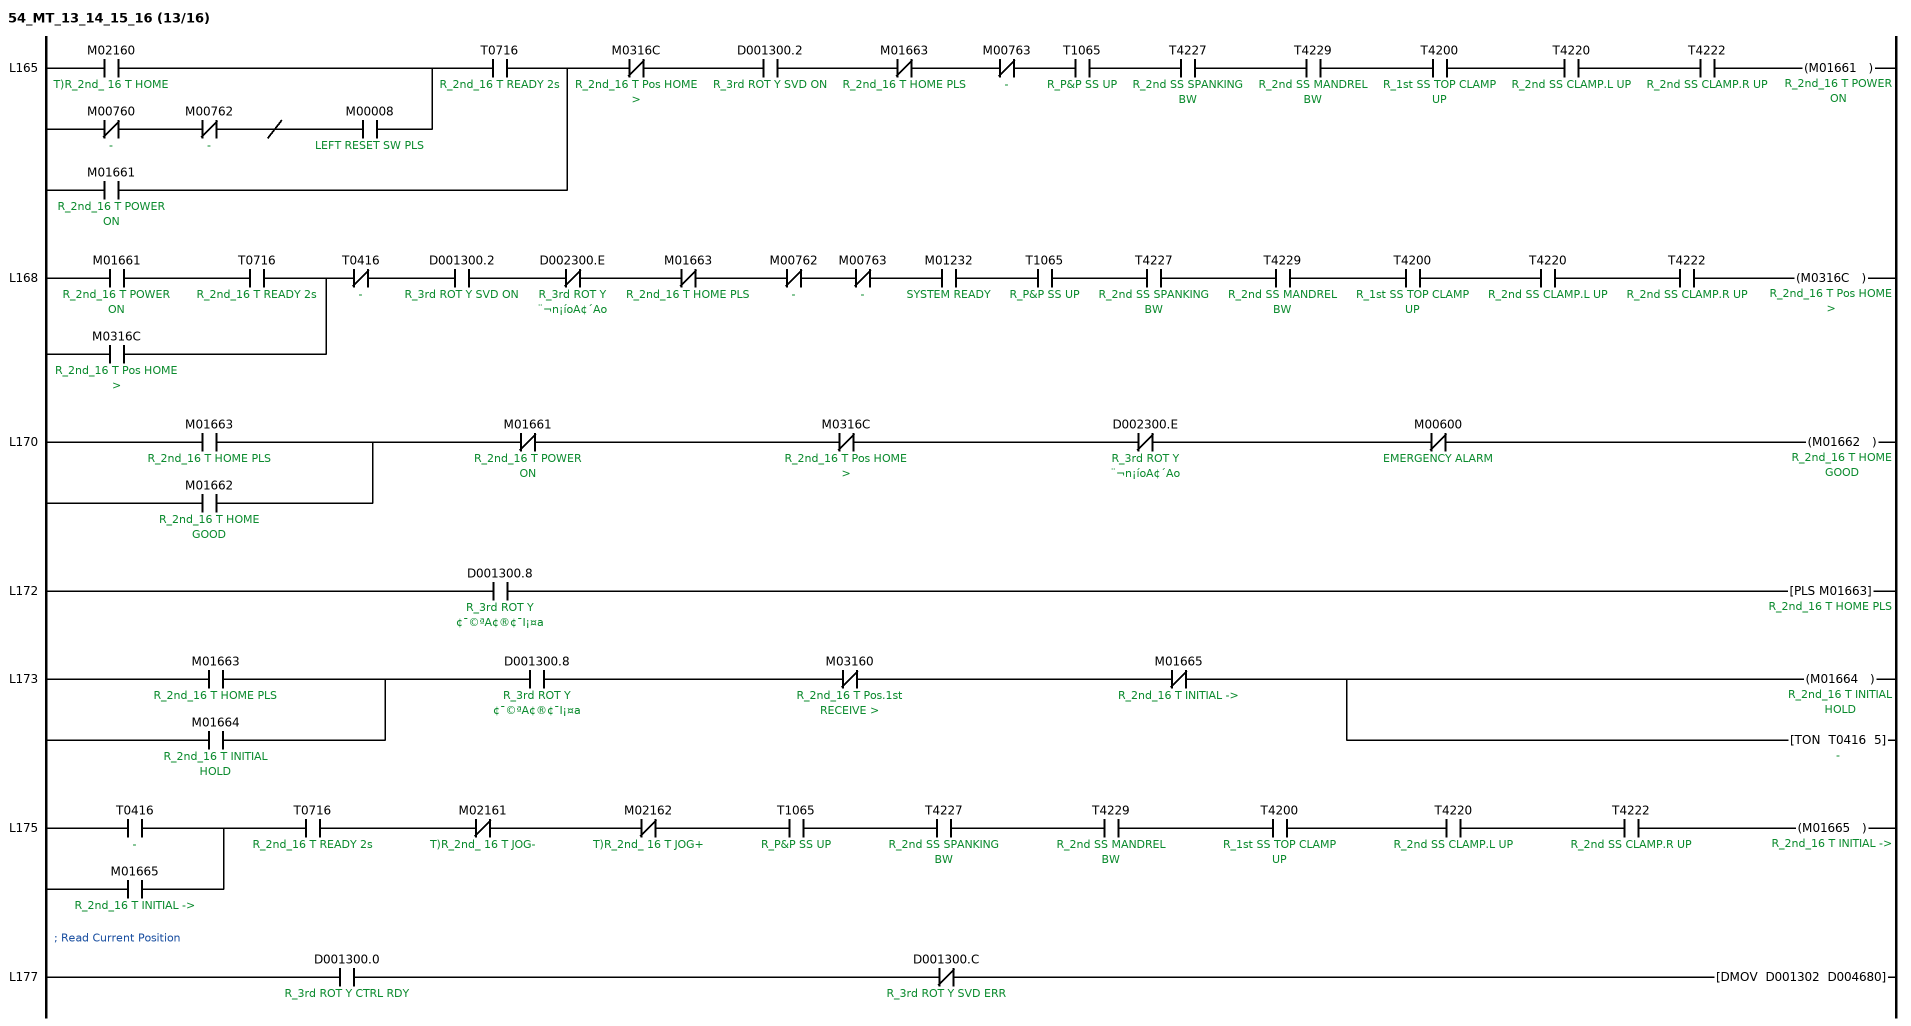
[picture p312: 54_MT_13_14_15_16 rungs L165-L177]
; L165
LOAD      M02160	// T)R_2nd_ 16 T HOME
LOAD NOT  M00760	// -
AND NOT   M00762	// -
NOT
AND       M00008	// LEFT RESET SW PLS
OR LOAD
AND       T0716	// R_2nd_16 T READY 2s
OR        M01661	// R_2nd_16 T POWER ON
AND NOT   M0316C	// R_2nd_16 T Pos HOME >
AND       D001300.2	// R_3rd ROT Y SVD ON
AND NOT   M01663	// R_2nd_16 T HOME PLS
AND NOT   M00763	// -
AND       T1065	// R_P&P SS UP
AND       T4227	// R_2nd SS SPANKING BW
AND       T4229	// R_2nd SS MANDREL BW
AND       T4200	// R_1st SS TOP CLAMP UP
AND       T4220	// R_2nd SS CLAMP.L UP
AND       T4222	// R_2nd SS CLAMP.R UP
OUT       M01661	// R_2nd_16 T POWER ON
; L168
LOAD      M01661	// R_2nd_16 T POWER ON
AND       T0716	// R_2nd_16 T READY 2s
OR        M0316C	// R_2nd_16 T Pos HOME >
AND NOT   T0416	// -
AND       D001300.2	// R_3rd ROT Y SVD ON
AND NOT   D002300.E	// R_3rd ROT Y ¨¬n¡íoA¢´Ao
AND NOT   M01663	// R_2nd_16 T HOME PLS
AND NOT   M00762	// -
AND NOT   M00763	// -
AND       M01232	// SYSTEM READY
AND       T1065	// R_P&P SS UP
AND       T4227	// R_2nd SS SPANKING BW
AND       T4229	// R_2nd SS MANDREL BW
AND       T4200	// R_1st SS TOP CLAMP UP
AND       T4220	// R_2nd SS CLAMP.L UP
AND       T4222	// R_2nd SS CLAMP.R UP
OUT       M0316C	// R_2nd_16 T Pos HOME >
; L170
LOAD      M01663	// R_2nd_16 T HOME PLS
OR        M01662	// R_2nd_16 T HOME GOOD
AND NOT   M01661	// R_2nd_16 T POWER ON
AND NOT   M0316C	// R_2nd_16 T Pos HOME >
AND NOT   D002300.E	// R_3rd ROT Y ¨¬n¡íoA¢´Ao
AND NOT   M00600	// EMERGENCY ALARM
OUT       M01662	// R_2nd_16 T HOME GOOD
; L172
LOAD      D001300.8	// R_3rd ROT Y ¢¯©ªA¢®¢¯I¡¤a
OUTP      M01663	// R_2nd_16 T HOME PLS
; L173
LOAD      M01663	// R_2nd_16 T HOME PLS
OR        M01664	// R_2nd_16 T INITIAL HOLD
AND       D001300.8	// R_3rd ROT Y ¢¯©ªA¢®¢¯I¡¤a
AND NOT   M03160	// R_2nd_16 T Pos.1st RECEIVE >
AND NOT   M01665	// R_2nd_16 T INITIAL ->
OUT       M01664	// R_2nd_16 T INITIAL HOLD
TON       T0416 5	// -
; L175
LOAD      T0416	// -
OR        M01665	// R_2nd_16 T INITIAL ->
AND       T0716	// R_2nd_16 T READY 2s
AND NOT   M02161	// T)R_2nd_ 16 T JOG-
AND NOT   M02162	// T)R_2nd_ 16 T JOG+
AND       T1065	// R_P&P SS UP
AND       T4227	// R_2nd SS SPANKING BW
AND       T4229	// R_2nd SS MANDREL BW
AND       T4200	// R_1st SS TOP CLAMP UP
AND       T4220	// R_2nd SS CLAMP.L UP
AND       T4222	// R_2nd SS CLAMP.R UP
OUT       M01665	// R_2nd_16 T INITIAL ->
; L177
LOAD      D001300.0	// R_3rd ROT Y CTRL RDY
AND NOT   D001300.C	// R_3rd ROT Y SVD ERR
DMOV      D001302 D004680
// output comment: Read Current Position

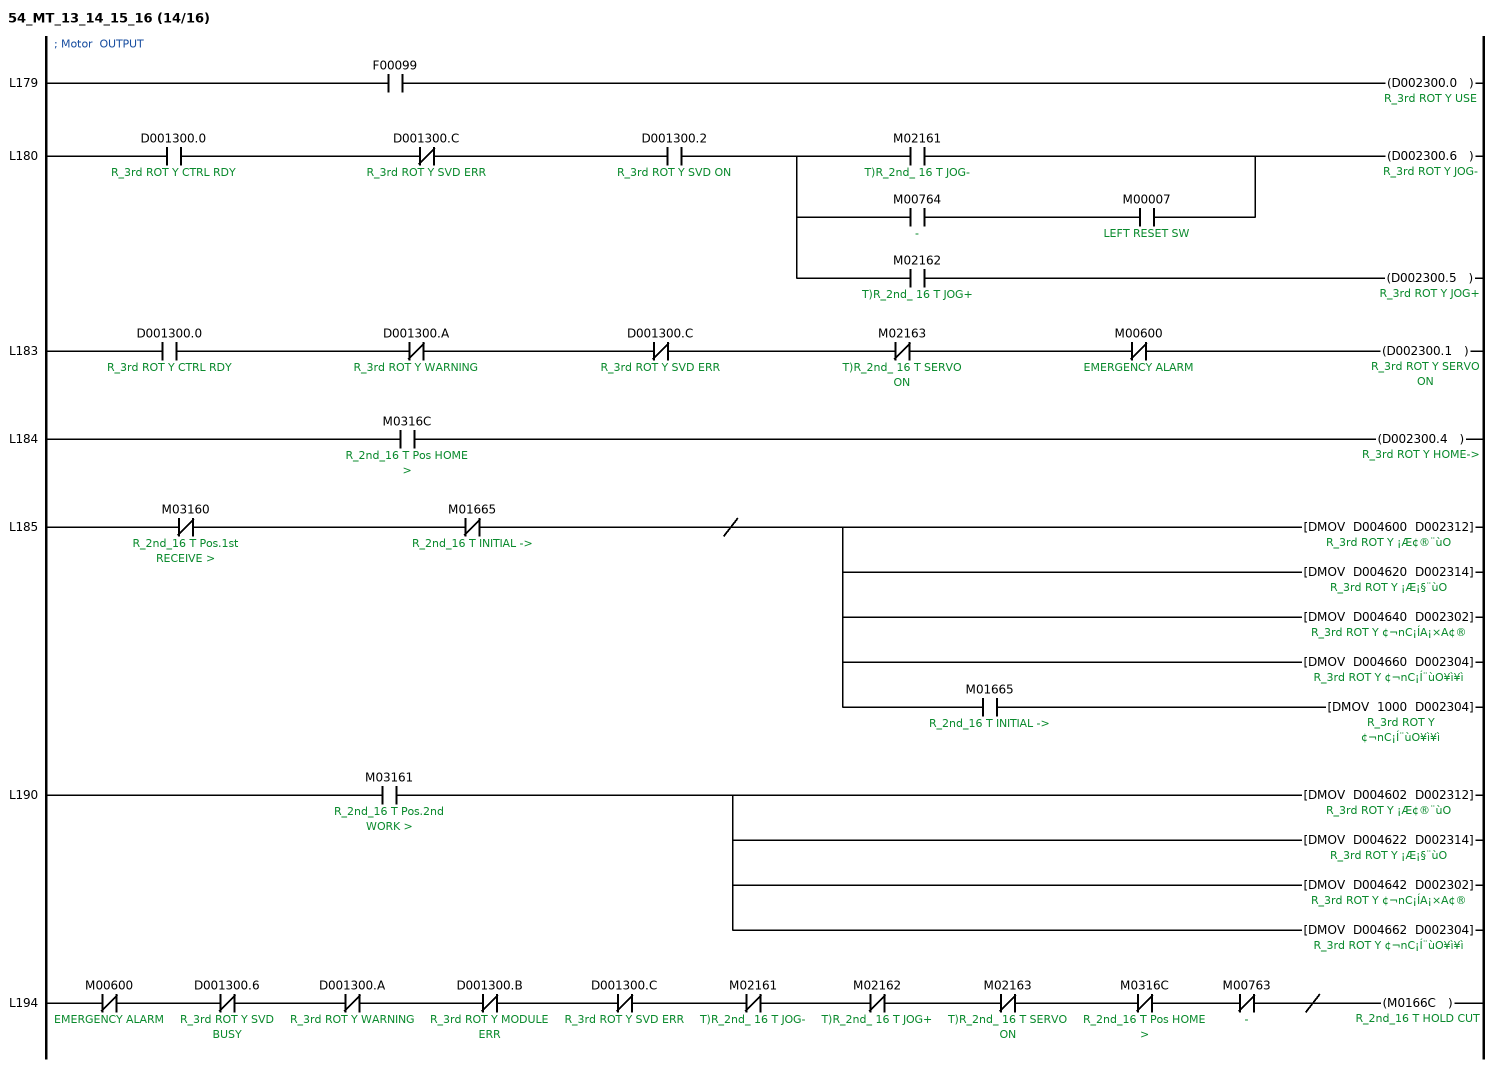
//  Motor  OUTPUT
; L179
LOAD      F00099
OUT       D002300.0	// R_3rd ROT Y USE
; L180
LOAD      D001300.0	// R_3rd ROT Y CTRL RDY
AND NOT   D001300.C	// R_3rd ROT Y SVD ERR
AND       D001300.2	// R_3rd ROT Y SVD ON
MPUSH
LOAD      M02161	// T)R_2nd_ 16 T JOG-
LOAD      M00764	// -
AND       M00007	// LEFT RESET SW
OR LOAD
AND LOAD
OUT       D002300.6	// R_3rd ROT Y JOG-
MPOP
AND       M02162	// T)R_2nd_ 16 T JOG+
OUT       D002300.5	// R_3rd ROT Y JOG+
; L183
LOAD      D001300.0	// R_3rd ROT Y CTRL RDY
AND NOT   D001300.A	// R_3rd ROT Y WARNING
AND NOT   D001300.C	// R_3rd ROT Y SVD ERR
AND NOT   M02163	// T)R_2nd_ 16 T SERVO ON
AND NOT   M00600	// EMERGENCY ALARM
OUT       D002300.1	// R_3rd ROT Y SERVO ON
; L184
LOAD      M0316C	// R_2nd_16 T Pos HOME >
OUT       D002300.4	// R_3rd ROT Y HOME->
; L185
LOAD NOT  M03160	// R_2nd_16 T Pos.1st RECEIVE >
AND NOT   M01665	// R_2nd_16 T INITIAL ->
NOT
DMOV      D004600 D002312	// R_3rd ROT Y ¡Æ¢®¨ùO
DMOV      D004620 D002314	// R_3rd ROT Y ¡Æ¡§¨ùO
DMOV      D004640 D002302	// R_3rd ROT Y ¢¬nC¡ÍA¡×A¢®
DMOV      D004660 D002304	// R_3rd ROT Y ¢¬nC¡Í¨ùO¥ì¥ì
AND       M01665	// R_2nd_16 T INITIAL ->
DMOV      1000 D002304	// R_3rd ROT Y ¢¬nC¡Í¨ùO¥ì¥ì
; L190
LOAD      M03161	// R_2nd_16 T Pos.2nd WORK >
DMOV      D004602 D002312	// R_3rd ROT Y ¡Æ¢®¨ùO
DMOV      D004622 D002314	// R_3rd ROT Y ¡Æ¡§¨ùO
DMOV      D004642 D002302	// R_3rd ROT Y ¢¬nC¡ÍA¡×A¢®
DMOV      D004662 D002304	// R_3rd ROT Y ¢¬nC¡Í¨ùO¥ì¥ì
; L194
LOAD NOT  M00600	// EMERGENCY ALARM
AND NOT   D001300.6	// R_3rd ROT Y SVD BUSY
AND NOT   D001300.A	// R_3rd ROT Y WARNING
AND NOT   D001300.B	// R_3rd ROT Y MODULE ERR
AND NOT   D001300.C	// R_3rd ROT Y SVD ERR
AND NOT   M02161	// T)R_2nd_ 16 T JOG-
AND NOT   M02162	// T)R_2nd_ 16 T JOG+
AND NOT   M02163	// T)R_2nd_ 16 T SERVO ON
AND NOT   M0316C	// R_2nd_16 T Pos HOME >
AND NOT   M00763	// -
NOT
OUT       M0166C	// R_2nd_16 T HOLD CUT

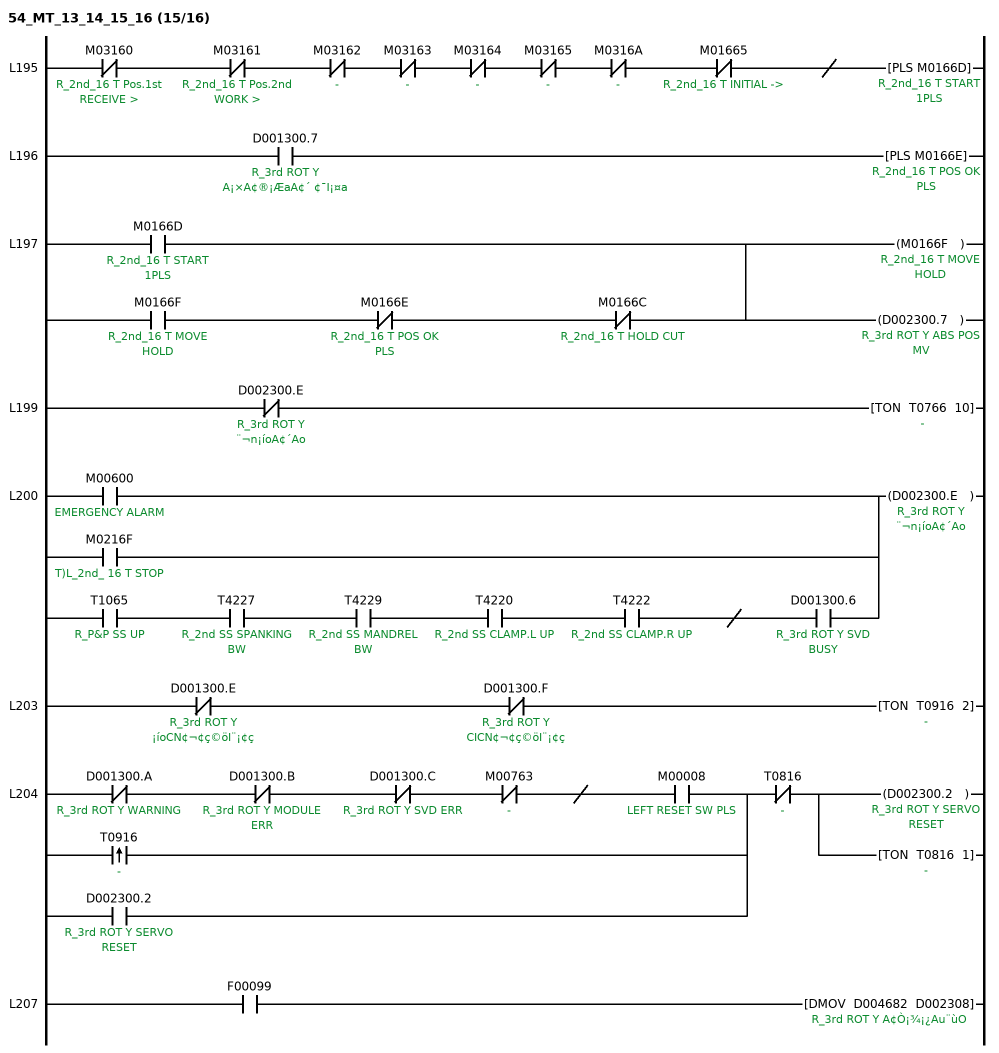
; L195
LOAD NOT  M03160	// R_2nd_16 T Pos.1st RECEIVE >
AND NOT   M03161	// R_2nd_16 T Pos.2nd WORK >
AND NOT   M03162	// -
AND NOT   M03163	// -
AND NOT   M03164	// -
AND NOT   M03165	// -
AND NOT   M0316A	// -
AND NOT   M01665	// R_2nd_16 T INITIAL ->
NOT
OUTP      M0166D	// R_2nd_16 T START 1PLS
; L196
LOAD      D001300.7	// R_3rd ROT Y A¡×A¢®¡ÆaA¢´ ¢¯I¡¤a
OUTP      M0166E	// R_2nd_16 T POS OK PLS
; L197
LOAD      M0166D	// R_2nd_16 T START 1PLS
LOAD      M0166F	// R_2nd_16 T MOVE HOLD
AND NOT   M0166E	// R_2nd_16 T POS OK PLS
AND NOT   M0166C	// R_2nd_16 T HOLD CUT
OR LOAD
OUT       M0166F	// R_2nd_16 T MOVE HOLD
OUT       D002300.7	// R_3rd ROT Y ABS POS MV
; L199
LOAD NOT  D002300.E	// R_3rd ROT Y ¨¬n¡íoA¢´Ao
TON       T0766 10	// -
; L200
LOAD      M00600	// EMERGENCY ALARM
OR        M0216F	// T)L_2nd_ 16 T STOP
LOAD      T1065	// R_P&P SS UP
AND       T4227	// R_2nd SS SPANKING BW
AND       T4229	// R_2nd SS MANDREL BW
AND       T4220	// R_2nd SS CLAMP.L UP
AND       T4222	// R_2nd SS CLAMP.R UP
NOT
AND       D001300.6	// R_3rd ROT Y SVD BUSY
OR LOAD
OUT       D002300.E	// R_3rd ROT Y ¨¬n¡íoA¢´Ao
; L203
LOAD NOT  D001300.E	// R_3rd ROT Y ¡íoCN¢¬¢ç©öI¨¡¢ç
AND NOT   D001300.F	// R_3rd ROT Y CICN¢¬¢ç©öI¨¡¢ç
TON       T0916 2	// -
; L204
LOAD NOT  D001300.A	// R_3rd ROT Y WARNING
AND NOT   D001300.B	// R_3rd ROT Y MODULE ERR
AND NOT   D001300.C	// R_3rd ROT Y SVD ERR
AND NOT   M00763	// -
NOT
AND       M00008	// LEFT RESET SW PLS
ORP       T0916	// -
OR        D002300.2	// R_3rd ROT Y SERVO RESET
AND NOT   T0816	// -
OUT       D002300.2	// R_3rd ROT Y SERVO RESET
TON       T0816 1	// -
; L207
LOAD      F00099
DMOV      D004682 D002308	// R_3rd ROT Y A¢Ò¡¾¡¿Au¨ùO

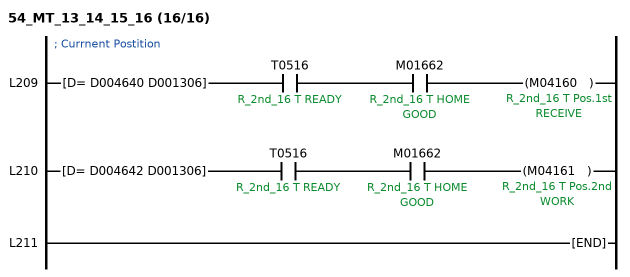
// Currnent Postition
; L209
LOADD=    D004640 D001306
AND       T0516	// R_2nd_16 T READY
AND       M01662	// R_2nd_16 T HOME GOOD
OUT       M04160	// R_2nd_16 T Pos.1st RECEIVE
; L210
LOADD=    D004642 D001306
AND       T0516	// R_2nd_16 T READY
AND       M01662	// R_2nd_16 T HOME GOOD
OUT       M04161	// R_2nd_16 T Pos.2nd WORK
; L211
END

PROGRAM 55_MT_17_18_19_20 (task: ¨ö¨¬A¥ì CA¡¤I¡¾¡¿¡¤¡Í)

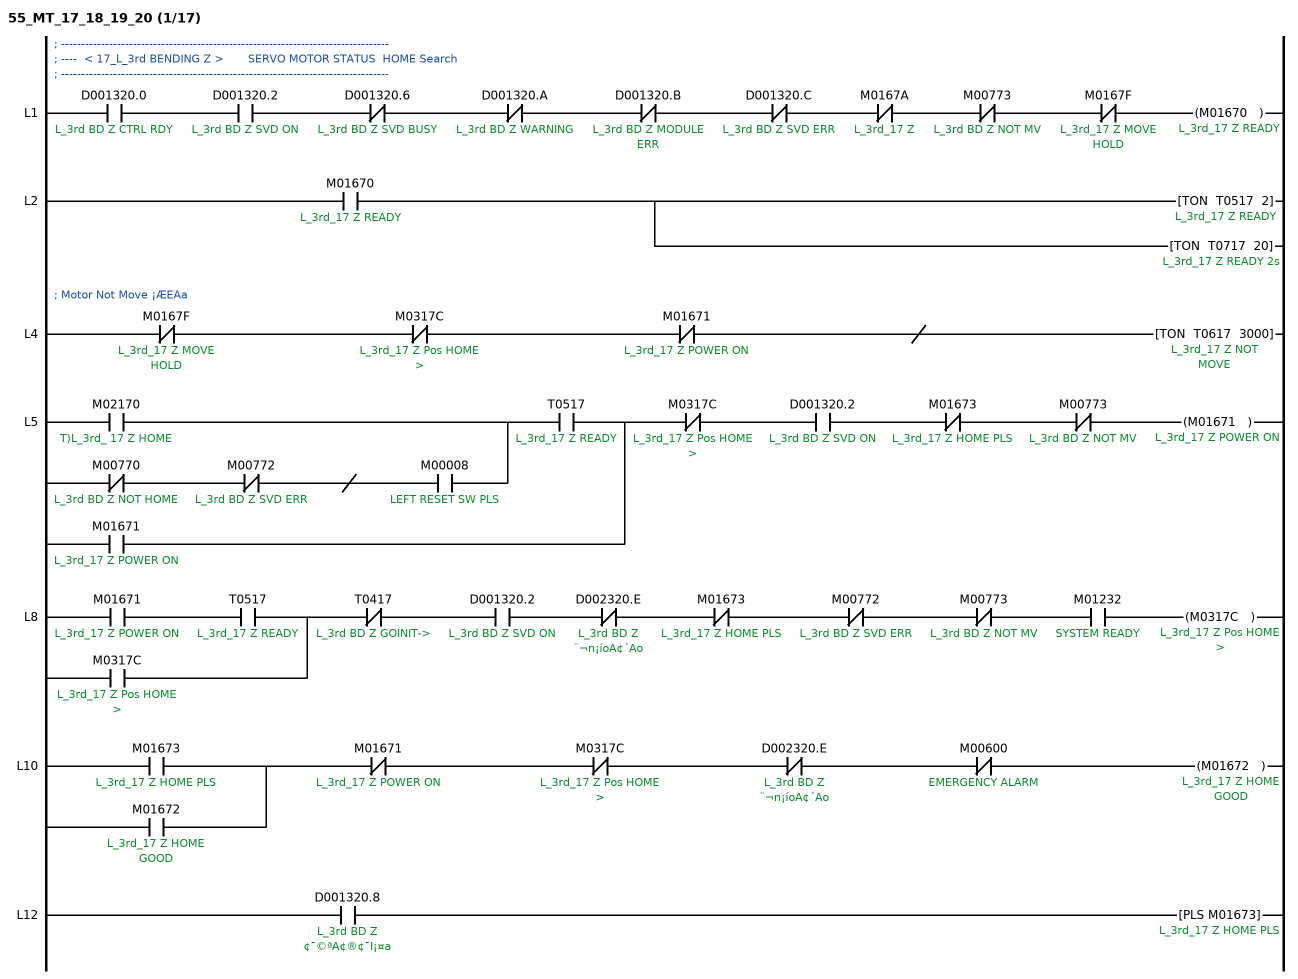
// ----------------------------------------------------------------------------------
// 
// ----  < 17_L_3rd BENDING Z >       SERVO MOTOR STATUS  HOME Search
// 
// ----------------------------------------------------------------------------------
; L1
LOAD      D001320.0	// L_3rd BD Z CTRL RDY
AND       D001320.2	// L_3rd BD Z SVD ON
AND NOT   D001320.6	// L_3rd BD Z SVD BUSY
AND NOT   D001320.A	// L_3rd BD Z WARNING
AND NOT   D001320.B	// L_3rd BD Z MODULE ERR
AND NOT   D001320.C	// L_3rd BD Z SVD ERR
AND NOT   M0167A	// L_3rd_17 Z
AND NOT   M00773	// L_3rd BD Z NOT MV
AND NOT   M0167F	// L_3rd_17 Z MOVE HOLD
OUT       M01670	// L_3rd_17 Z READY
; L2
LOAD      M01670	// L_3rd_17 Z READY
TON       T0517 2	// L_3rd_17 Z READY
TON       T0717 20	// L_3rd_17 Z READY 2s
; L4
LOAD NOT  M0167F	// L_3rd_17 Z MOVE HOLD
AND NOT   M0317C	// L_3rd_17 Z Pos HOME >
AND NOT   M01671	// L_3rd_17 Z POWER ON
NOT
TON       T0617 3000	// L_3rd_17 Z NOT MOVE
// output comment: Motor Not Move ¡ÆEAa
; L5
LOAD      M02170	// T)L_3rd_ 17 Z HOME
LOAD NOT  M00770	// L_3rd BD Z NOT HOME
AND NOT   M00772	// L_3rd BD Z SVD ERR
NOT
AND       M00008	// LEFT RESET SW PLS
OR LOAD
AND       T0517	// L_3rd_17 Z READY
OR        M01671	// L_3rd_17 Z POWER ON
AND NOT   M0317C	// L_3rd_17 Z Pos HOME >
AND       D001320.2	// L_3rd BD Z SVD ON
AND NOT   M01673	// L_3rd_17 Z HOME PLS
AND NOT   M00773	// L_3rd BD Z NOT MV
OUT       M01671	// L_3rd_17 Z POWER ON
; L8
LOAD      M01671	// L_3rd_17 Z POWER ON
AND       T0517	// L_3rd_17 Z READY
OR        M0317C	// L_3rd_17 Z Pos HOME >
AND NOT   T0417	// L_3rd BD Z GOINIT->
AND       D001320.2	// L_3rd BD Z SVD ON
AND NOT   D002320.E	// L_3rd BD Z ¨¬n¡íoA¢´Ao
AND NOT   M01673	// L_3rd_17 Z HOME PLS
AND NOT   M00772	// L_3rd BD Z SVD ERR
AND NOT   M00773	// L_3rd BD Z NOT MV
AND       M01232	// SYSTEM READY
OUT       M0317C	// L_3rd_17 Z Pos HOME >
; L10
LOAD      M01673	// L_3rd_17 Z HOME PLS
OR        M01672	// L_3rd_17 Z HOME GOOD
AND NOT   M01671	// L_3rd_17 Z POWER ON
AND NOT   M0317C	// L_3rd_17 Z Pos HOME >
AND NOT   D002320.E	// L_3rd BD Z ¨¬n¡íoA¢´Ao
AND NOT   M00600	// EMERGENCY ALARM
OUT       M01672	// L_3rd_17 Z HOME GOOD
; L12
LOAD      D001320.8	// L_3rd BD Z ¢¯©ªA¢®¢¯I¡¤a
OUTP      M01673	// L_3rd_17 Z HOME PLS

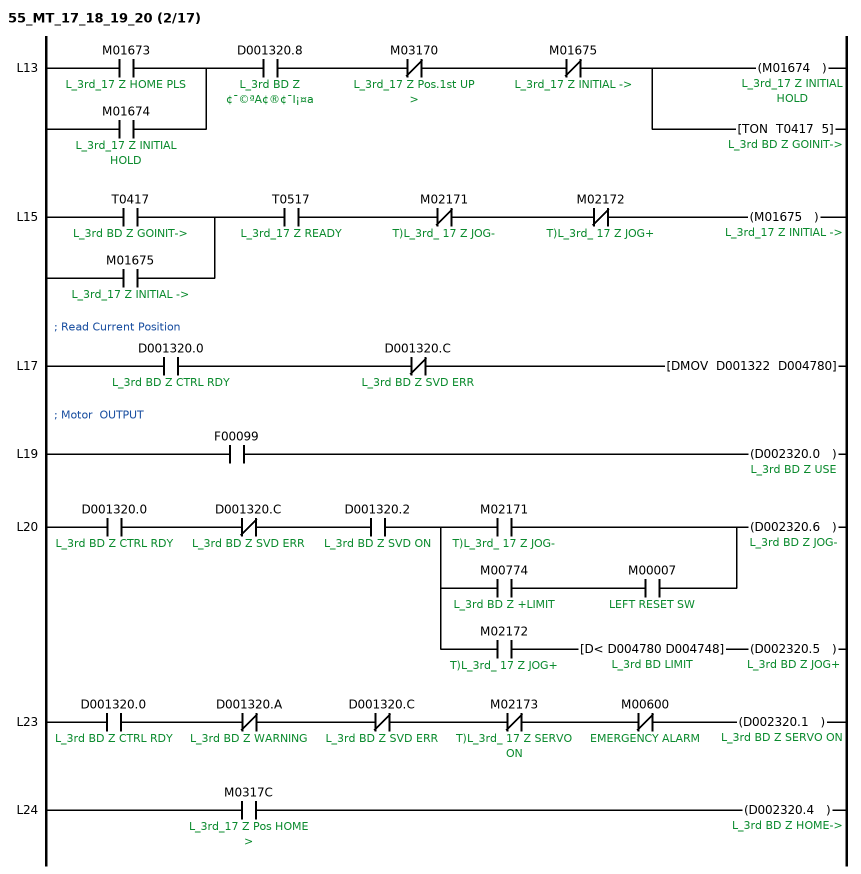
; L13
LOAD      M01673	// L_3rd_17 Z HOME PLS
OR        M01674	// L_3rd_17 Z INITIAL HOLD
AND       D001320.8	// L_3rd BD Z ¢¯©ªA¢®¢¯I¡¤a
AND NOT   M03170	// L_3rd_17 Z Pos.1st UP >
AND NOT   M01675	// L_3rd_17 Z INITIAL ->
OUT       M01674	// L_3rd_17 Z INITIAL HOLD
TON       T0417 5	// L_3rd BD Z GOINIT->
; L15
LOAD      T0417	// L_3rd BD Z GOINIT->
OR        M01675	// L_3rd_17 Z INITIAL ->
AND       T0517	// L_3rd_17 Z READY
AND NOT   M02171	// T)L_3rd_ 17 Z JOG-
AND NOT   M02172	// T)L_3rd_ 17 Z JOG+
OUT       M01675	// L_3rd_17 Z INITIAL ->
; L17
LOAD      D001320.0	// L_3rd BD Z CTRL RDY
AND NOT   D001320.C	// L_3rd BD Z SVD ERR
DMOV      D001322 D004780
// output comment: Read Current Position
//  Motor  OUTPUT
; L19
LOAD      F00099
OUT       D002320.0	// L_3rd BD Z USE
; L20
LOAD      D001320.0	// L_3rd BD Z CTRL RDY
AND NOT   D001320.C	// L_3rd BD Z SVD ERR
AND       D001320.2	// L_3rd BD Z SVD ON
MPUSH
LOAD      M02171	// T)L_3rd_ 17 Z JOG-
LOAD      M00774	// L_3rd BD Z +LIMIT
AND       M00007	// LEFT RESET SW
OR LOAD
AND LOAD
OUT       D002320.6	// L_3rd BD Z JOG-
MPOP
AND       M02172	// T)L_3rd_ 17 Z JOG+
ANDD<     D004780 D004748	// L_3rd BD LIMIT
OUT       D002320.5	// L_3rd BD Z JOG+
; L23
LOAD      D001320.0	// L_3rd BD Z CTRL RDY
AND NOT   D001320.A	// L_3rd BD Z WARNING
AND NOT   D001320.C	// L_3rd BD Z SVD ERR
AND NOT   M02173	// T)L_3rd_ 17 Z SERVO ON
AND NOT   M00600	// EMERGENCY ALARM
OUT       D002320.1	// L_3rd BD Z SERVO ON
; L24
LOAD      M0317C	// L_3rd_17 Z Pos HOME >
OUT       D002320.4	// L_3rd BD Z HOME->

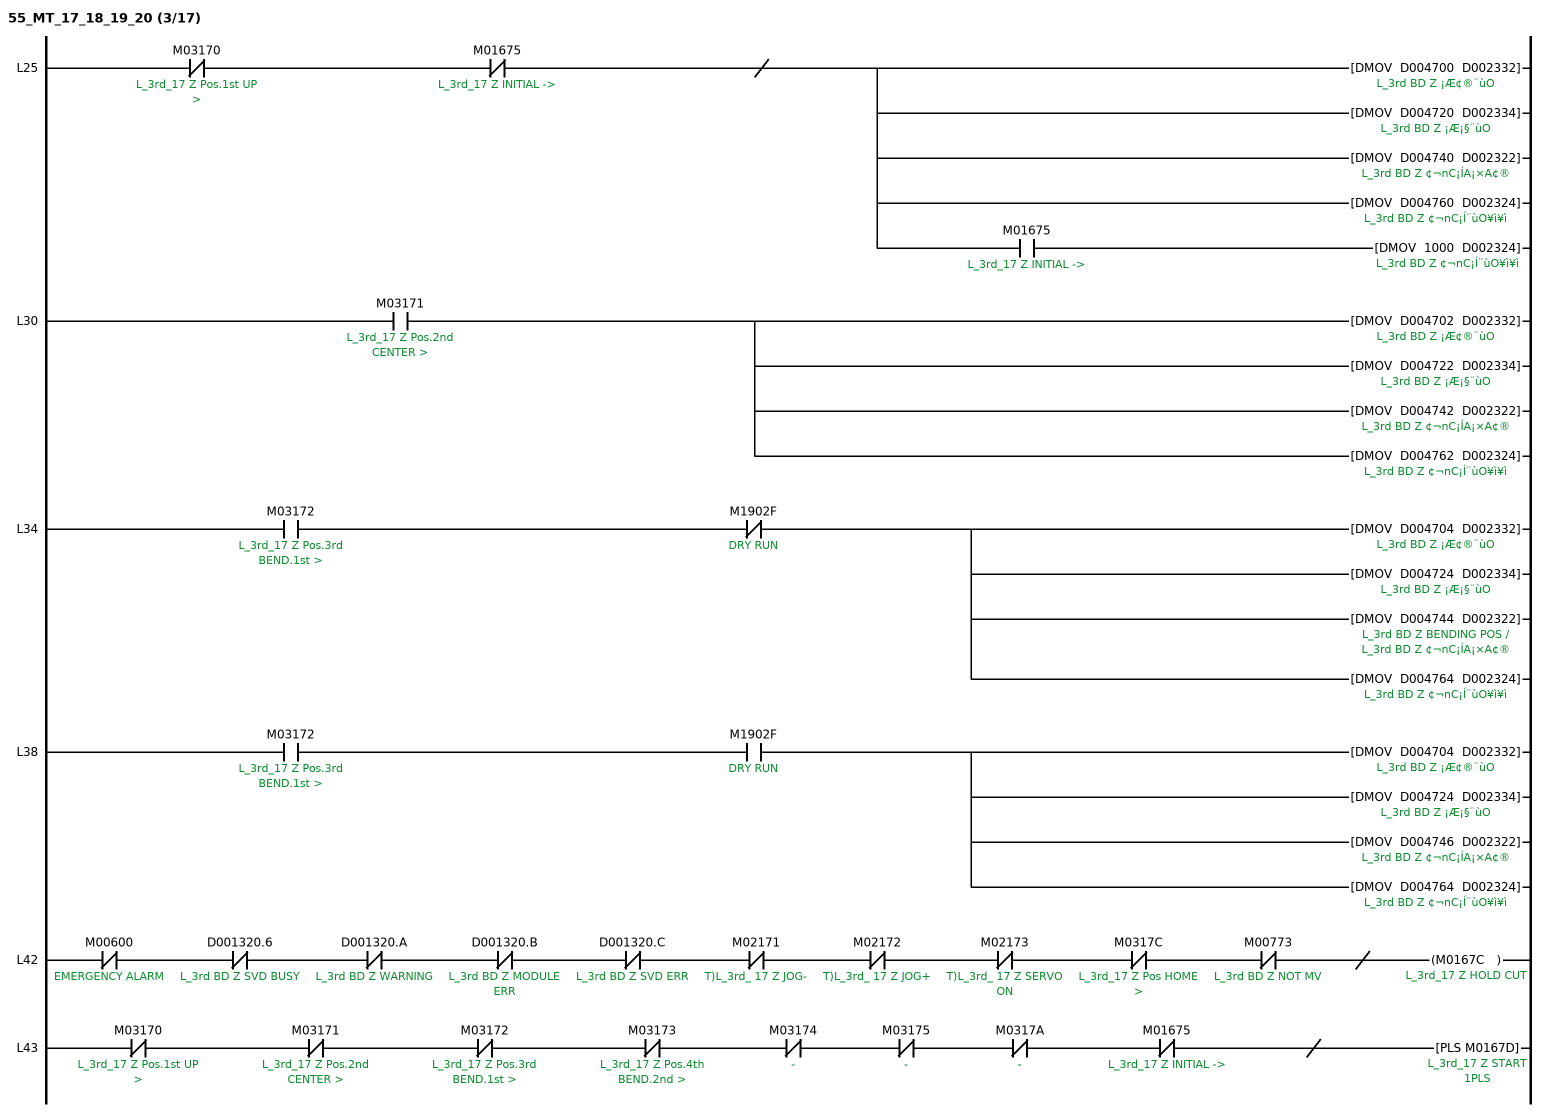
; L25
LOAD NOT  M03170	// L_3rd_17 Z Pos.1st UP >
AND NOT   M01675	// L_3rd_17 Z INITIAL ->
NOT
DMOV      D004700 D002332	// L_3rd BD Z ¡Æ¢®¨ùO
DMOV      D004720 D002334	// L_3rd BD Z ¡Æ¡§¨ùO
DMOV      D004740 D002322	// L_3rd BD Z ¢¬nC¡ÍA¡×A¢®
DMOV      D004760 D002324	// L_3rd BD Z ¢¬nC¡Í¨ùO¥ì¥ì
AND       M01675	// L_3rd_17 Z INITIAL ->
DMOV      1000 D002324	// L_3rd BD Z ¢¬nC¡Í¨ùO¥ì¥ì
; L30
LOAD      M03171	// L_3rd_17 Z Pos.2nd CENTER >
DMOV      D004702 D002332	// L_3rd BD Z ¡Æ¢®¨ùO
DMOV      D004722 D002334	// L_3rd BD Z ¡Æ¡§¨ùO
DMOV      D004742 D002322	// L_3rd BD Z ¢¬nC¡ÍA¡×A¢®
DMOV      D004762 D002324	// L_3rd BD Z ¢¬nC¡Í¨ùO¥ì¥ì
; L34
LOAD      M03172	// L_3rd_17 Z Pos.3rd BEND.1st >
AND NOT   M1902F	// DRY RUN
DMOV      D004704 D002332	// L_3rd BD Z ¡Æ¢®¨ùO
DMOV      D004724 D002334	// L_3rd BD Z ¡Æ¡§¨ùO
DMOV      D004744 D002322	// L_3rd BD Z BENDING POS / L_3rd BD Z ¢¬nC¡ÍA¡×A¢®
DMOV      D004764 D002324	// L_3rd BD Z ¢¬nC¡Í¨ùO¥ì¥ì
; L38
LOAD      M03172	// L_3rd_17 Z Pos.3rd BEND.1st >
AND       M1902F	// DRY RUN
DMOV      D004704 D002332	// L_3rd BD Z ¡Æ¢®¨ùO
DMOV      D004724 D002334	// L_3rd BD Z ¡Æ¡§¨ùO
DMOV      D004746 D002322	// L_3rd BD Z ¢¬nC¡ÍA¡×A¢®
DMOV      D004764 D002324	// L_3rd BD Z ¢¬nC¡Í¨ùO¥ì¥ì
; L42
LOAD NOT  M00600	// EMERGENCY ALARM
AND NOT   D001320.6	// L_3rd BD Z SVD BUSY
AND NOT   D001320.A	// L_3rd BD Z WARNING
AND NOT   D001320.B	// L_3rd BD Z MODULE ERR
AND NOT   D001320.C	// L_3rd BD Z SVD ERR
AND NOT   M02171	// T)L_3rd_ 17 Z JOG-
AND NOT   M02172	// T)L_3rd_ 17 Z JOG+
AND NOT   M02173	// T)L_3rd_ 17 Z SERVO ON
AND NOT   M0317C	// L_3rd_17 Z Pos HOME >
AND NOT   M00773	// L_3rd BD Z NOT MV
NOT
OUT       M0167C	// L_3rd_17 Z HOLD CUT
; L43
LOAD NOT  M03170	// L_3rd_17 Z Pos.1st UP >
AND NOT   M03171	// L_3rd_17 Z Pos.2nd CENTER >
AND NOT   M03172	// L_3rd_17 Z Pos.3rd BEND.1st >
AND NOT   M03173	// L_3rd_17 Z Pos.4th BEND.2nd >
AND NOT   M03174	// -
AND NOT   M03175	// -
AND NOT   M0317A	// -
AND NOT   M01675	// L_3rd_17 Z INITIAL ->
NOT
OUTP      M0167D	// L_3rd_17 Z START 1PLS

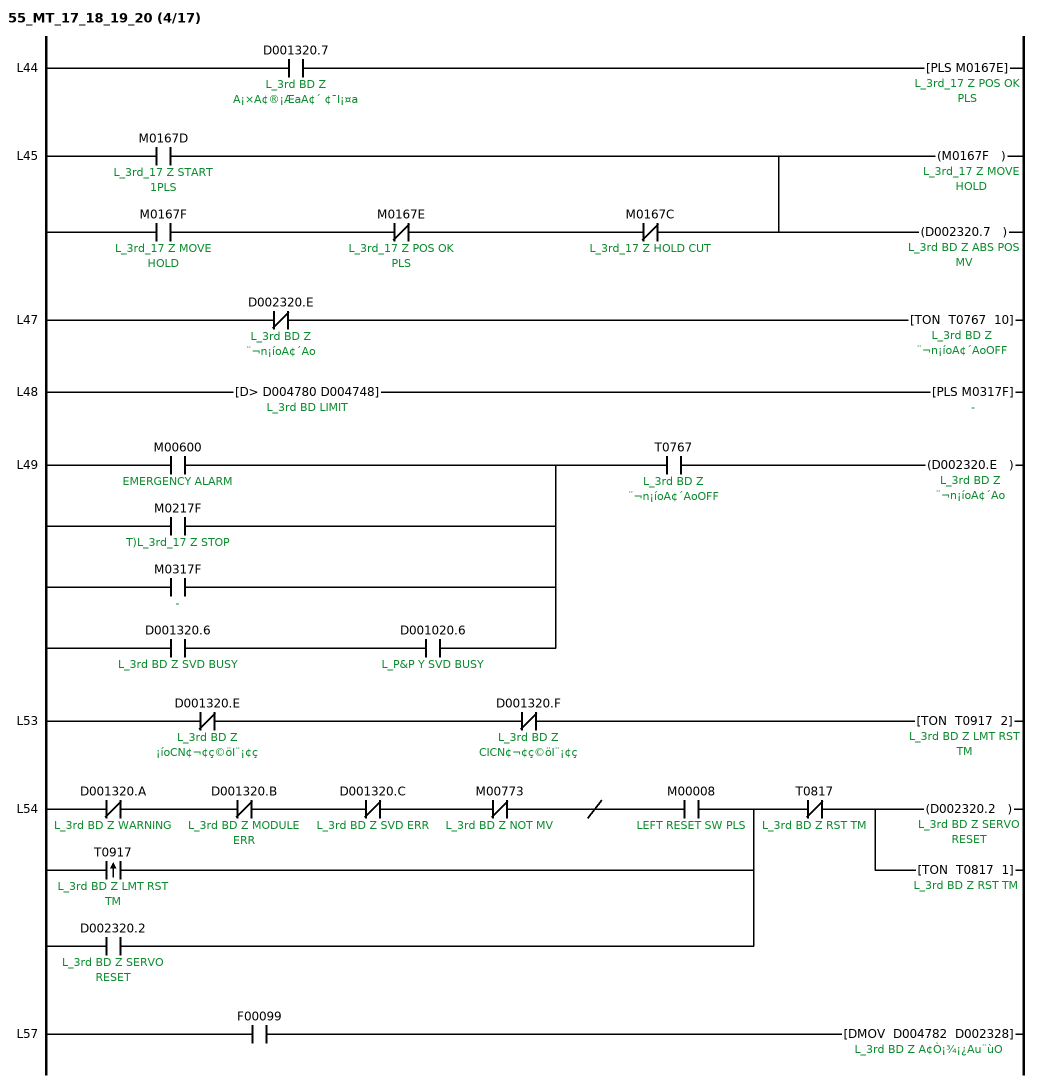
; L44
LOAD      D001320.7	// L_3rd BD Z A¡×A¢®¡ÆaA¢´ ¢¯I¡¤a
OUTP      M0167E	// L_3rd_17 Z POS OK PLS
; L45
LOAD      M0167D	// L_3rd_17 Z START 1PLS
LOAD      M0167F	// L_3rd_17 Z MOVE HOLD
AND NOT   M0167E	// L_3rd_17 Z POS OK PLS
AND NOT   M0167C	// L_3rd_17 Z HOLD CUT
OR LOAD
OUT       M0167F	// L_3rd_17 Z MOVE HOLD
OUT       D002320.7	// L_3rd BD Z ABS POS MV
; L47
LOAD NOT  D002320.E	// L_3rd BD Z ¨¬n¡íoA¢´Ao
TON       T0767 10	// L_3rd BD Z ¨¬n¡íoA¢´AoOFF
; L48
LOADD>    D004780 D004748	// L_3rd BD LIMIT
OUTP      M0317F	// -
; L49
LOAD      M00600	// EMERGENCY ALARM
OR        M0217F	// T)L_3rd_17 Z STOP
OR        M0317F	// -
LOAD      D001320.6	// L_3rd BD Z SVD BUSY
AND       D001020.6	// L_P&P Y SVD BUSY
OR LOAD
AND       T0767	// L_3rd BD Z ¨¬n¡íoA¢´AoOFF
OUT       D002320.E	// L_3rd BD Z ¨¬n¡íoA¢´Ao
; L53
LOAD NOT  D001320.E	// L_3rd BD Z ¡íoCN¢¬¢ç©öI¨¡¢ç
AND NOT   D001320.F	// L_3rd BD Z CICN¢¬¢ç©öI¨¡¢ç
TON       T0917 2	// L_3rd BD Z LMT RST TM
; L54
LOAD NOT  D001320.A	// L_3rd BD Z WARNING
AND NOT   D001320.B	// L_3rd BD Z MODULE ERR
AND NOT   D001320.C	// L_3rd BD Z SVD ERR
AND NOT   M00773	// L_3rd BD Z NOT MV
NOT
AND       M00008	// LEFT RESET SW PLS
ORP       T0917	// L_3rd BD Z LMT RST TM
OR        D002320.2	// L_3rd BD Z SERVO RESET
AND NOT   T0817	// L_3rd BD Z RST TM
OUT       D002320.2	// L_3rd BD Z SERVO RESET
TON       T0817 1	// L_3rd BD Z RST TM
; L57
LOAD      F00099
DMOV      D004782 D002328	// L_3rd BD Z A¢Ò¡¾¡¿Au¨ùO

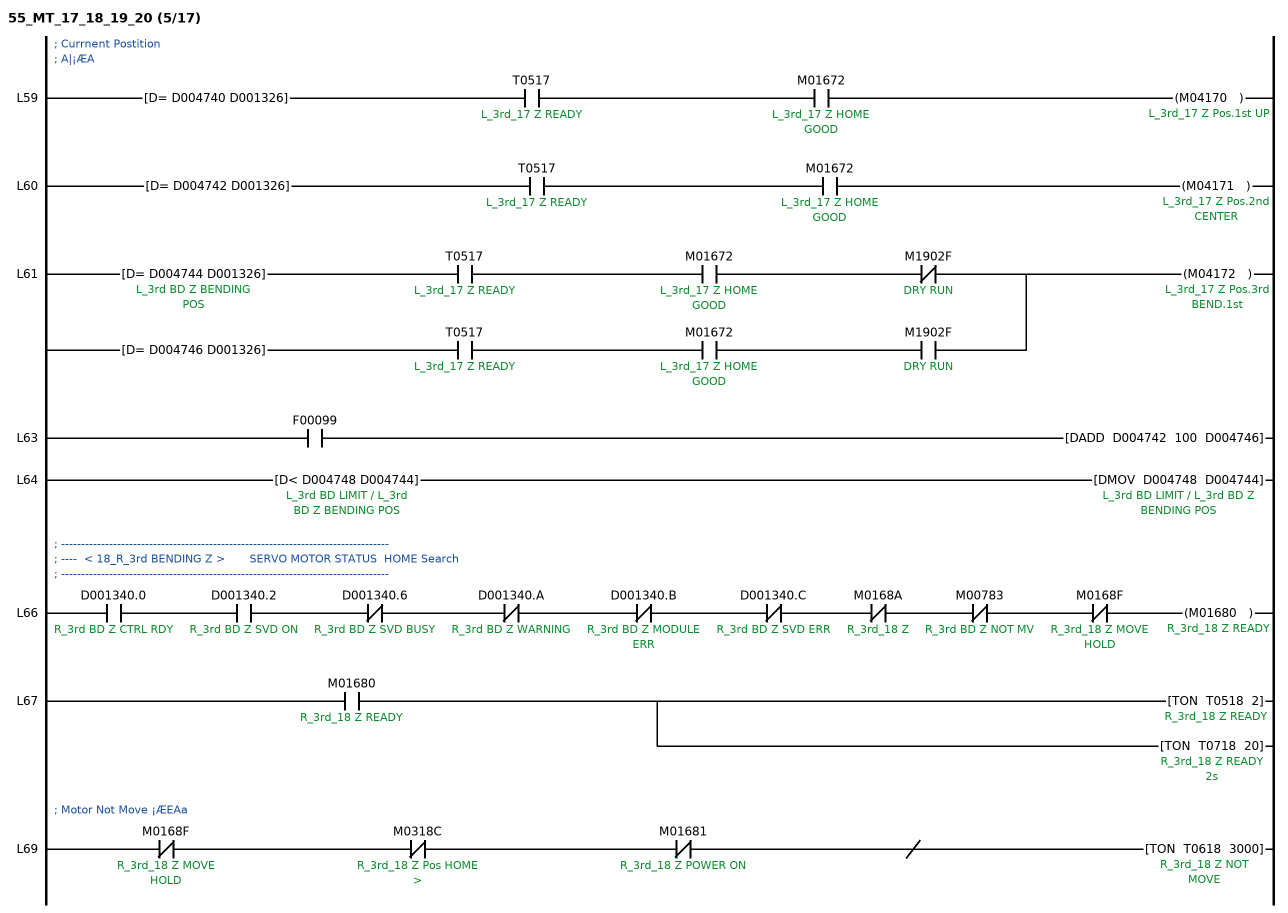
// Currnent Postition
; L59
LOADD=    D004740 D001326
AND       T0517	// L_3rd_17 Z READY
AND       M01672	// L_3rd_17 Z HOME GOOD
OUT       M04170	// L_3rd_17 Z Pos.1st UP
// output comment: A|¡ÆA
; L60
LOADD=    D004742 D001326
AND       T0517	// L_3rd_17 Z READY
AND       M01672	// L_3rd_17 Z HOME GOOD
OUT       M04171	// L_3rd_17 Z Pos.2nd CENTER
; L61
LOADD=    D004744 D001326	// L_3rd BD Z BENDING POS
AND       T0517	// L_3rd_17 Z READY
AND       M01672	// L_3rd_17 Z HOME GOOD
AND NOT   M1902F	// DRY RUN
LOADD=    D004746 D001326
AND       T0517	// L_3rd_17 Z READY
AND       M01672	// L_3rd_17 Z HOME GOOD
AND       M1902F	// DRY RUN
OR LOAD
OUT       M04172	// L_3rd_17 Z Pos.3rd BEND.1st
; L63
LOAD      F00099
DADD      D004742 100 D004746
; L64
LOADD<    D004748 D004744	// L_3rd BD LIMIT / L_3rd BD Z BENDING POS
DMOV      D004748 D004744	// L_3rd BD LIMIT / L_3rd BD Z BENDING POS
// ----------------------------------------------------------------------------------
// 
// ----  < 18_R_3rd BENDING Z >       SERVO MOTOR STATUS  HOME Search
// 
// ----------------------------------------------------------------------------------
; L66
LOAD      D001340.0	// R_3rd BD Z CTRL RDY
AND       D001340.2	// R_3rd BD Z SVD ON
AND NOT   D001340.6	// R_3rd BD Z SVD BUSY
AND NOT   D001340.A	// R_3rd BD Z WARNING
AND NOT   D001340.B	// R_3rd BD Z MODULE ERR
AND NOT   D001340.C	// R_3rd BD Z SVD ERR
AND NOT   M0168A	// R_3rd_18 Z
AND NOT   M00783	// R_3rd BD Z NOT MV
AND NOT   M0168F	// R_3rd_18 Z MOVE HOLD
OUT       M01680	// R_3rd_18 Z READY
; L67
LOAD      M01680	// R_3rd_18 Z READY
TON       T0518 2	// R_3rd_18 Z READY
TON       T0718 20	// R_3rd_18 Z READY 2s
; L69
LOAD NOT  M0168F	// R_3rd_18 Z MOVE HOLD
AND NOT   M0318C	// R_3rd_18 Z Pos HOME >
AND NOT   M01681	// R_3rd_18 Z POWER ON
NOT
TON       T0618 3000	// R_3rd_18 Z NOT MOVE
// output comment: Motor Not Move ¡ÆEAa

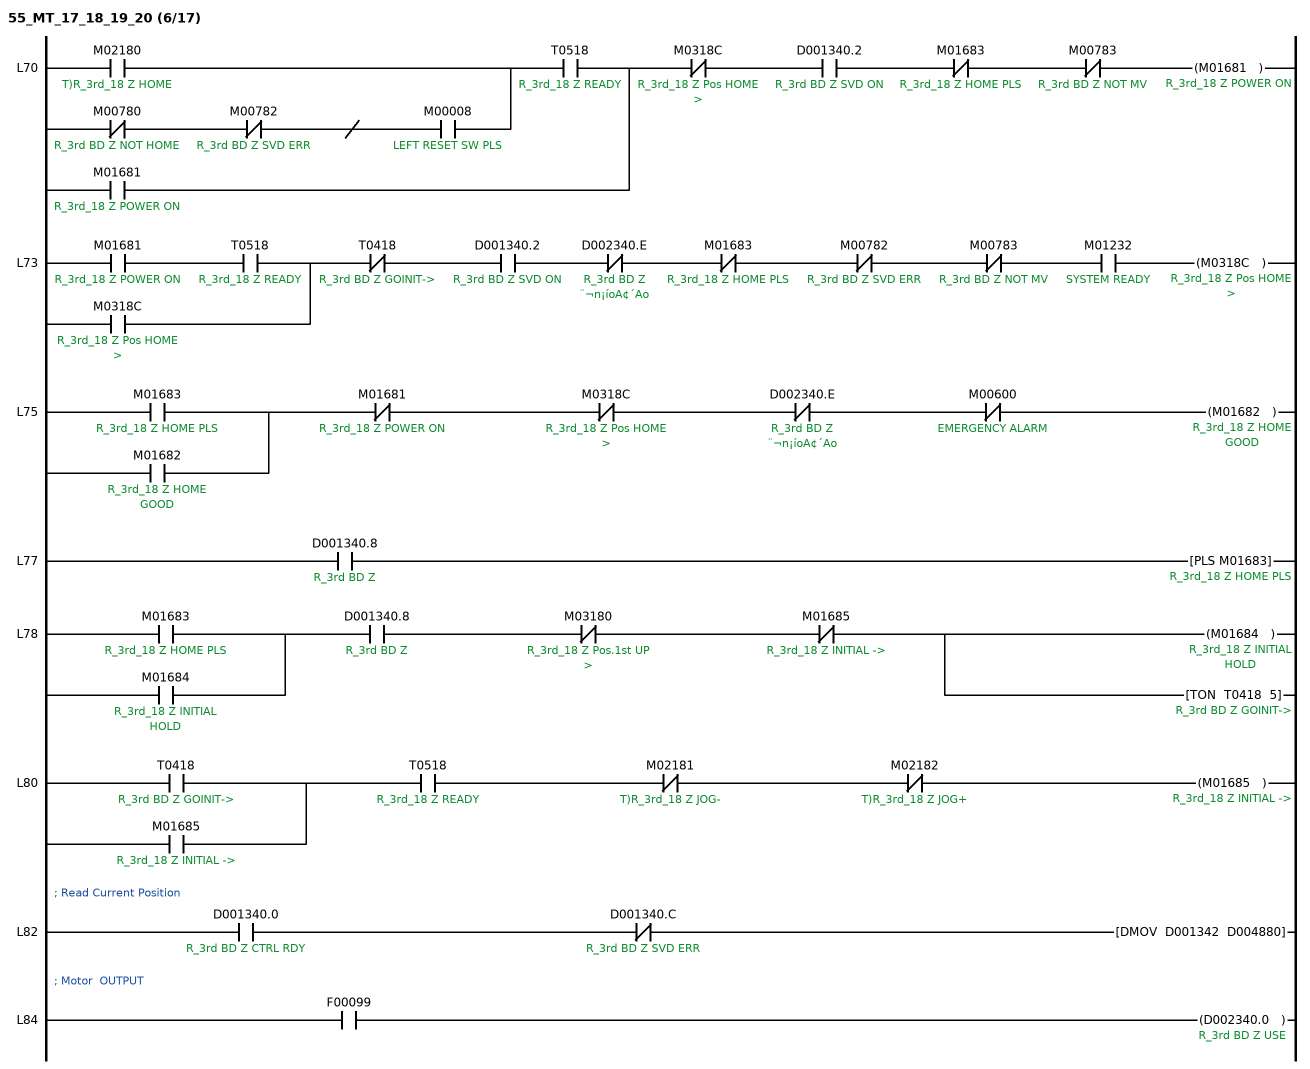
; L70
LOAD      M02180	// T)R_3rd_18 Z HOME
LOAD NOT  M00780	// R_3rd BD Z NOT HOME
AND NOT   M00782	// R_3rd BD Z SVD ERR
NOT
AND       M00008	// LEFT RESET SW PLS
OR LOAD
AND       T0518	// R_3rd_18 Z READY
OR        M01681	// R_3rd_18 Z POWER ON
AND NOT   M0318C	// R_3rd_18 Z Pos HOME >
AND       D001340.2	// R_3rd BD Z SVD ON
AND NOT   M01683	// R_3rd_18 Z HOME PLS
AND NOT   M00783	// R_3rd BD Z NOT MV
OUT       M01681	// R_3rd_18 Z POWER ON
; L73
LOAD      M01681	// R_3rd_18 Z POWER ON
AND       T0518	// R_3rd_18 Z READY
OR        M0318C	// R_3rd_18 Z Pos HOME >
AND NOT   T0418	// R_3rd BD Z GOINIT->
AND       D001340.2	// R_3rd BD Z SVD ON
AND NOT   D002340.E	// R_3rd BD Z ¨¬n¡íoA¢´Ao
AND NOT   M01683	// R_3rd_18 Z HOME PLS
AND NOT   M00782	// R_3rd BD Z SVD ERR
AND NOT   M00783	// R_3rd BD Z NOT MV
AND       M01232	// SYSTEM READY
OUT       M0318C	// R_3rd_18 Z Pos HOME >
; L75
LOAD      M01683	// R_3rd_18 Z HOME PLS
OR        M01682	// R_3rd_18 Z HOME GOOD
AND NOT   M01681	// R_3rd_18 Z POWER ON
AND NOT   M0318C	// R_3rd_18 Z Pos HOME >
AND NOT   D002340.E	// R_3rd BD Z ¨¬n¡íoA¢´Ao
AND NOT   M00600	// EMERGENCY ALARM
OUT       M01682	// R_3rd_18 Z HOME GOOD
; L77
LOAD      D001340.8	// R_3rd BD Z
OUTP      M01683	// R_3rd_18 Z HOME PLS
; L78
LOAD      M01683	// R_3rd_18 Z HOME PLS
OR        M01684	// R_3rd_18 Z INITIAL HOLD
AND       D001340.8	// R_3rd BD Z
AND NOT   M03180	// R_3rd_18 Z Pos.1st UP >
AND NOT   M01685	// R_3rd_18 Z INITIAL ->
OUT       M01684	// R_3rd_18 Z INITIAL HOLD
TON       T0418 5	// R_3rd BD Z GOINIT->
; L80
LOAD      T0418	// R_3rd BD Z GOINIT->
OR        M01685	// R_3rd_18 Z INITIAL ->
AND       T0518	// R_3rd_18 Z READY
AND NOT   M02181	// T)R_3rd_18 Z JOG-
AND NOT   M02182	// T)R_3rd_18 Z JOG+
OUT       M01685	// R_3rd_18 Z INITIAL ->
; L82
LOAD      D001340.0	// R_3rd BD Z CTRL RDY
AND NOT   D001340.C	// R_3rd BD Z SVD ERR
DMOV      D001342 D004880
// output comment: Read Current Position
//  Motor  OUTPUT
; L84
LOAD      F00099
OUT       D002340.0	// R_3rd BD Z USE

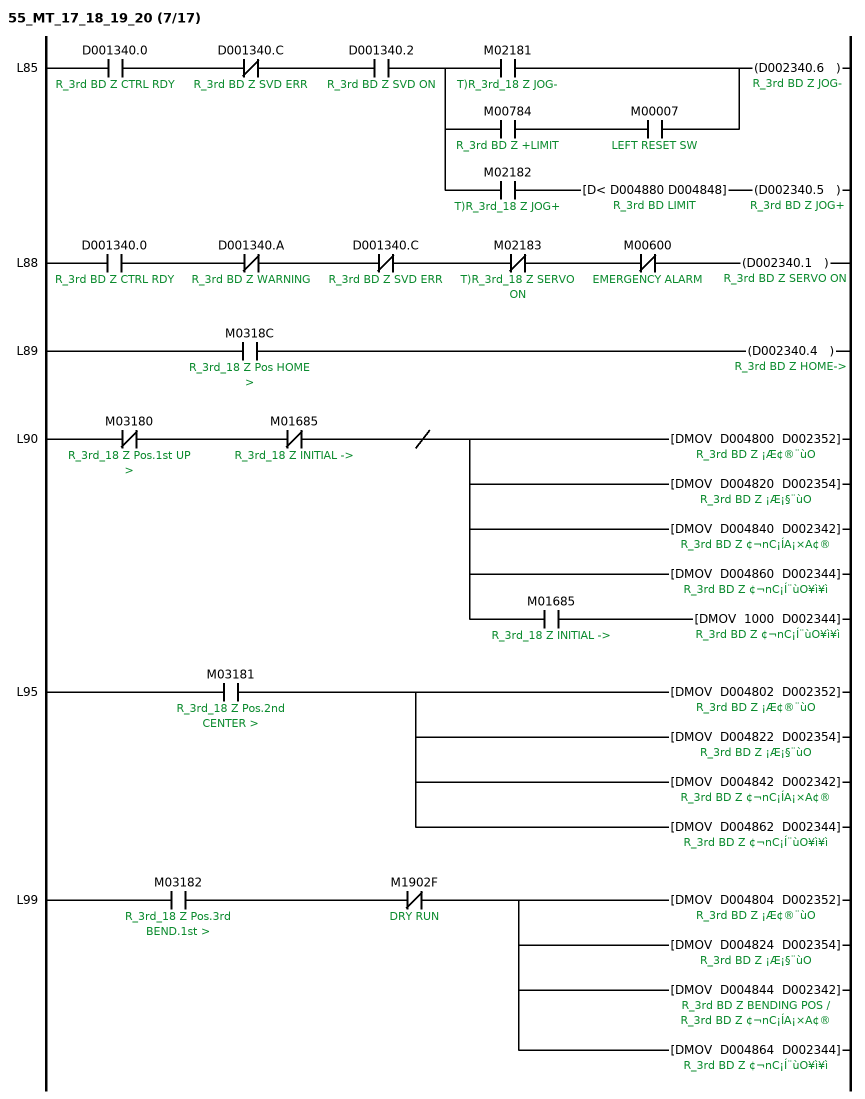
; L85
LOAD      D001340.0	// R_3rd BD Z CTRL RDY
AND NOT   D001340.C	// R_3rd BD Z SVD ERR
AND       D001340.2	// R_3rd BD Z SVD ON
MPUSH
LOAD      M02181	// T)R_3rd_18 Z JOG-
LOAD      M00784	// R_3rd BD Z +LIMIT
AND       M00007	// LEFT RESET SW
OR LOAD
AND LOAD
OUT       D002340.6	// R_3rd BD Z JOG-
MPOP
AND       M02182	// T)R_3rd_18 Z JOG+
ANDD<     D004880 D004848	// R_3rd BD LIMIT
OUT       D002340.5	// R_3rd BD Z JOG+
; L88
LOAD      D001340.0	// R_3rd BD Z CTRL RDY
AND NOT   D001340.A	// R_3rd BD Z WARNING
AND NOT   D001340.C	// R_3rd BD Z SVD ERR
AND NOT   M02183	// T)R_3rd_18 Z SERVO ON
AND NOT   M00600	// EMERGENCY ALARM
OUT       D002340.1	// R_3rd BD Z SERVO ON
; L89
LOAD      M0318C	// R_3rd_18 Z Pos HOME >
OUT       D002340.4	// R_3rd BD Z HOME->
; L90
LOAD NOT  M03180	// R_3rd_18 Z Pos.1st UP >
AND NOT   M01685	// R_3rd_18 Z INITIAL ->
NOT
DMOV      D004800 D002352	// R_3rd BD Z ¡Æ¢®¨ùO
DMOV      D004820 D002354	// R_3rd BD Z ¡Æ¡§¨ùO
DMOV      D004840 D002342	// R_3rd BD Z ¢¬nC¡ÍA¡×A¢®
DMOV      D004860 D002344	// R_3rd BD Z ¢¬nC¡Í¨ùO¥ì¥ì
AND       M01685	// R_3rd_18 Z INITIAL ->
DMOV      1000 D002344	// R_3rd BD Z ¢¬nC¡Í¨ùO¥ì¥ì
; L95
LOAD      M03181	// R_3rd_18 Z Pos.2nd CENTER >
DMOV      D004802 D002352	// R_3rd BD Z ¡Æ¢®¨ùO
DMOV      D004822 D002354	// R_3rd BD Z ¡Æ¡§¨ùO
DMOV      D004842 D002342	// R_3rd BD Z ¢¬nC¡ÍA¡×A¢®
DMOV      D004862 D002344	// R_3rd BD Z ¢¬nC¡Í¨ùO¥ì¥ì
; L99
LOAD      M03182	// R_3rd_18 Z Pos.3rd BEND.1st >
AND NOT   M1902F	// DRY RUN
DMOV      D004804 D002352	// R_3rd BD Z ¡Æ¢®¨ùO
DMOV      D004824 D002354	// R_3rd BD Z ¡Æ¡§¨ùO
DMOV      D004844 D002342	// R_3rd BD Z BENDING POS / R_3rd BD Z ¢¬nC¡ÍA¡×A¢®
DMOV      D004864 D002344	// R_3rd BD Z ¢¬nC¡Í¨ùO¥ì¥ì

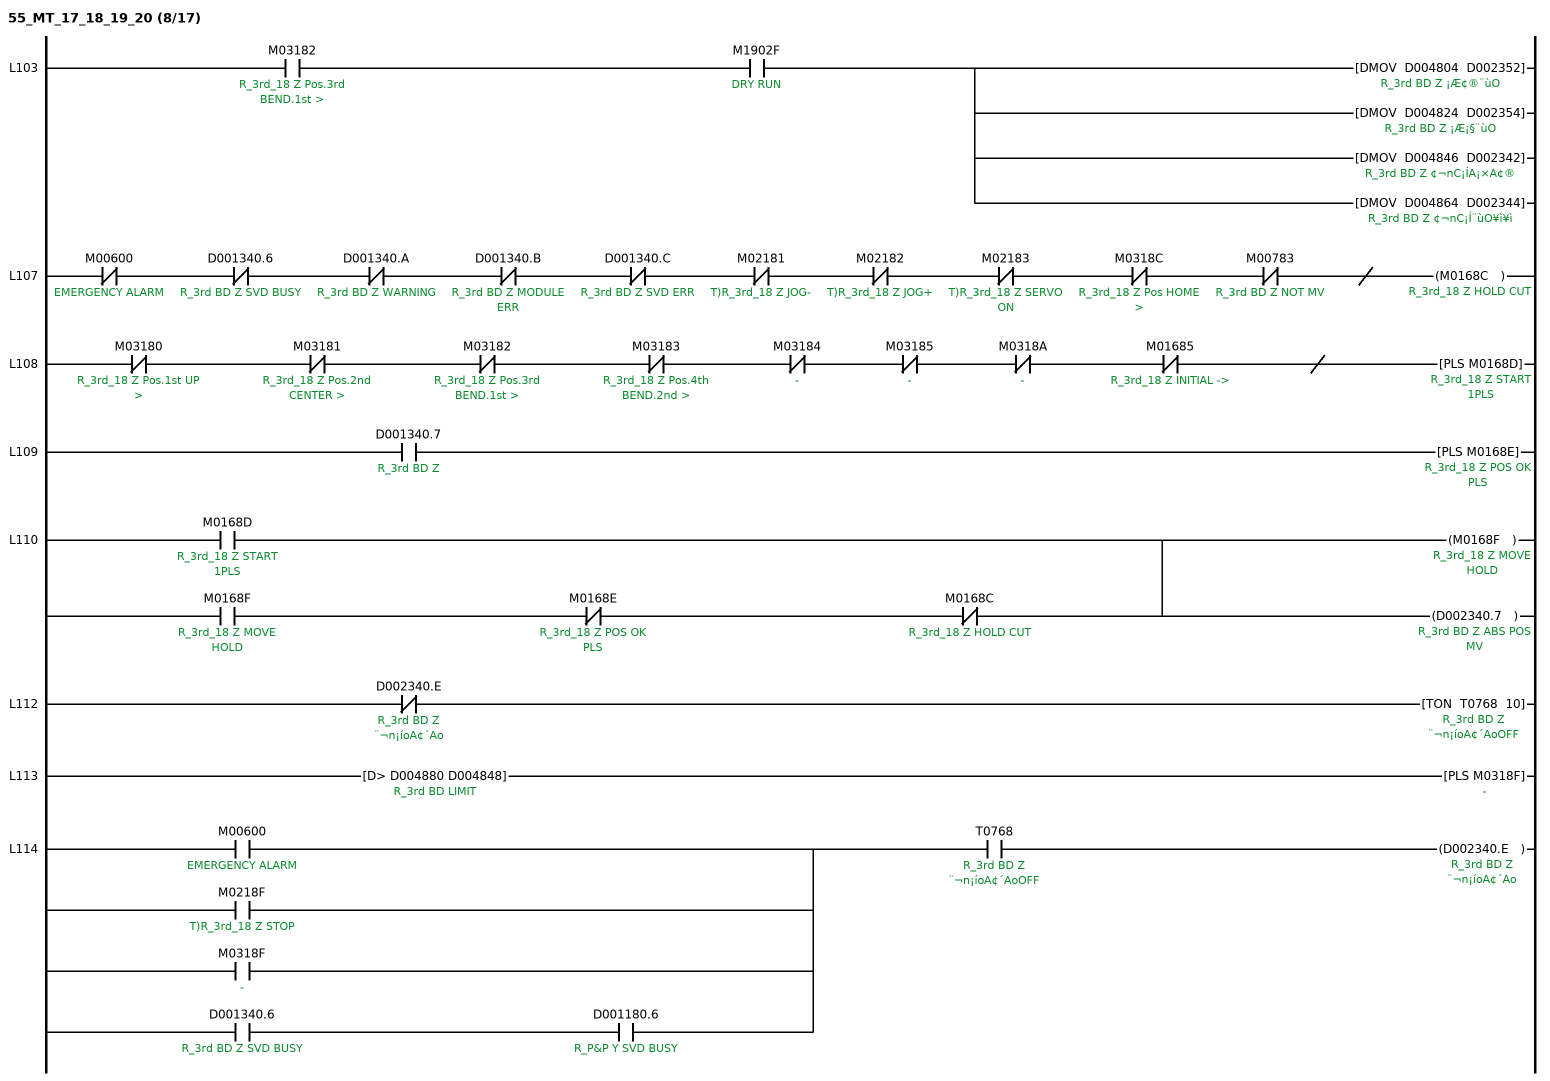
; L103
LOAD      M03182	// R_3rd_18 Z Pos.3rd BEND.1st >
AND       M1902F	// DRY RUN
DMOV      D004804 D002352	// R_3rd BD Z ¡Æ¢®¨ùO
DMOV      D004824 D002354	// R_3rd BD Z ¡Æ¡§¨ùO
DMOV      D004846 D002342	// R_3rd BD Z ¢¬nC¡ÍA¡×A¢®
DMOV      D004864 D002344	// R_3rd BD Z ¢¬nC¡Í¨ùO¥ì¥ì
; L107
LOAD NOT  M00600	// EMERGENCY ALARM
AND NOT   D001340.6	// R_3rd BD Z SVD BUSY
AND NOT   D001340.A	// R_3rd BD Z WARNING
AND NOT   D001340.B	// R_3rd BD Z MODULE ERR
AND NOT   D001340.C	// R_3rd BD Z SVD ERR
AND NOT   M02181	// T)R_3rd_18 Z JOG-
AND NOT   M02182	// T)R_3rd_18 Z JOG+
AND NOT   M02183	// T)R_3rd_18 Z SERVO ON
AND NOT   M0318C	// R_3rd_18 Z Pos HOME >
AND NOT   M00783	// R_3rd BD Z NOT MV
NOT
OUT       M0168C	// R_3rd_18 Z HOLD CUT
; L108
LOAD NOT  M03180	// R_3rd_18 Z Pos.1st UP >
AND NOT   M03181	// R_3rd_18 Z Pos.2nd CENTER >
AND NOT   M03182	// R_3rd_18 Z Pos.3rd BEND.1st >
AND NOT   M03183	// R_3rd_18 Z Pos.4th BEND.2nd >
AND NOT   M03184	// -
AND NOT   M03185	// -
AND NOT   M0318A	// -
AND NOT   M01685	// R_3rd_18 Z INITIAL ->
NOT
OUTP      M0168D	// R_3rd_18 Z START 1PLS
; L109
LOAD      D001340.7	// R_3rd BD Z
OUTP      M0168E	// R_3rd_18 Z POS OK PLS
; L110
LOAD      M0168D	// R_3rd_18 Z START 1PLS
LOAD      M0168F	// R_3rd_18 Z MOVE HOLD
AND NOT   M0168E	// R_3rd_18 Z POS OK PLS
AND NOT   M0168C	// R_3rd_18 Z HOLD CUT
OR LOAD
OUT       M0168F	// R_3rd_18 Z MOVE HOLD
OUT       D002340.7	// R_3rd BD Z ABS POS MV
; L112
LOAD NOT  D002340.E	// R_3rd BD Z ¨¬n¡íoA¢´Ao
TON       T0768 10	// R_3rd BD Z ¨¬n¡íoA¢´AoOFF
; L113
LOADD>    D004880 D004848	// R_3rd BD LIMIT
OUTP      M0318F	// -
; L114
LOAD      M00600	// EMERGENCY ALARM
OR        M0218F	// T)R_3rd_18 Z STOP
OR        M0318F	// -
LOAD      D001340.6	// R_3rd BD Z SVD BUSY
AND       D001180.6	// R_P&P Y SVD BUSY
OR LOAD
AND       T0768	// R_3rd BD Z ¨¬n¡íoA¢´AoOFF
OUT       D002340.E	// R_3rd BD Z ¨¬n¡íoA¢´Ao

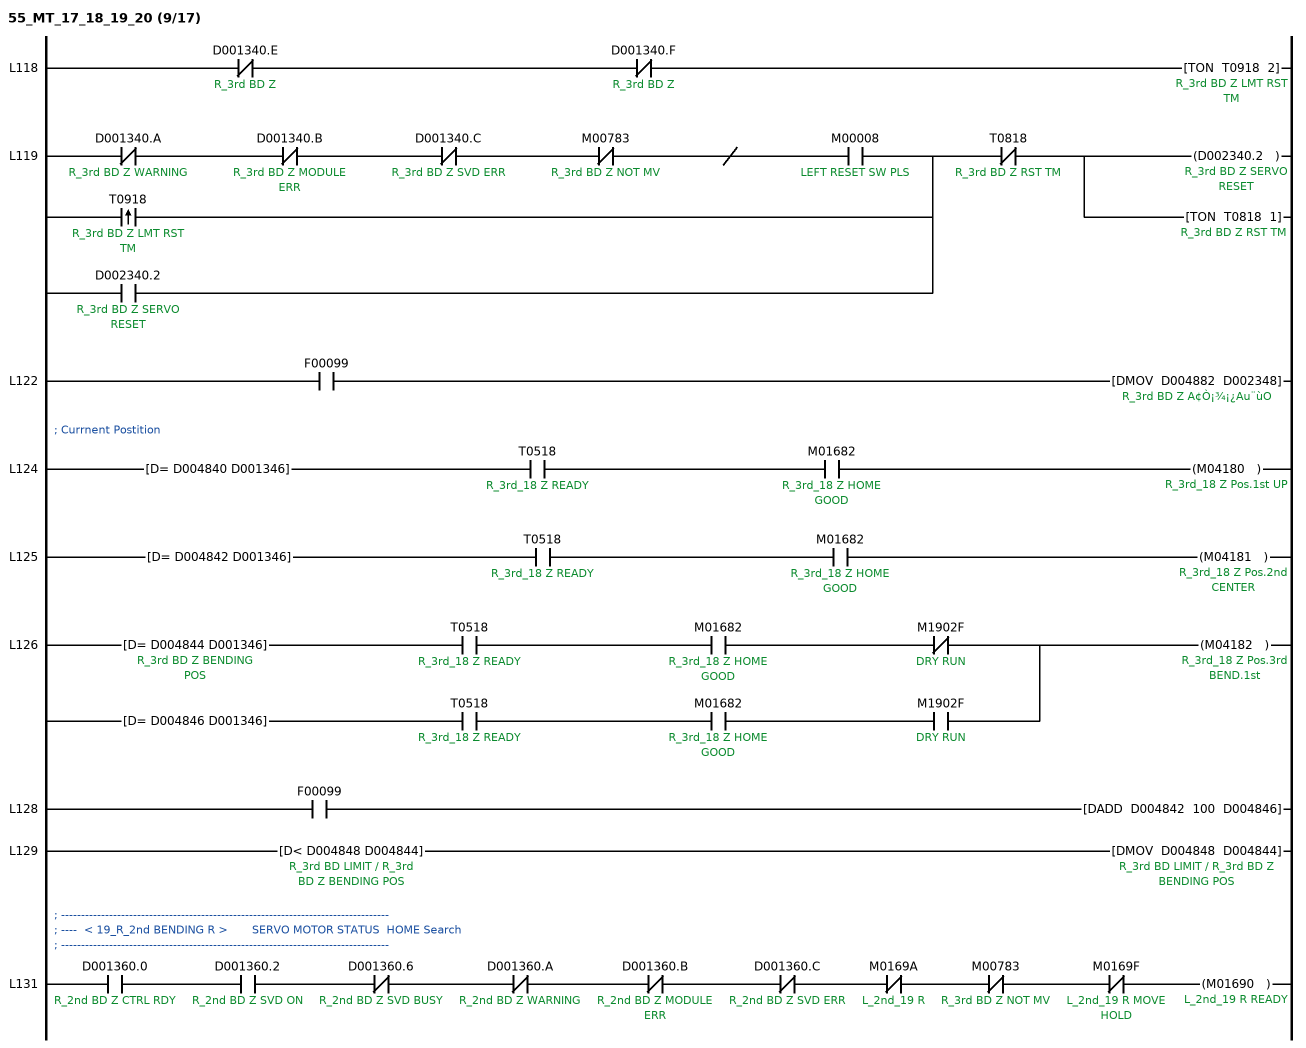
; L118
LOAD NOT  D001340.E	// R_3rd BD Z
AND NOT   D001340.F	// R_3rd BD Z
TON       T0918 2	// R_3rd BD Z LMT RST TM
; L119
LOAD NOT  D001340.A	// R_3rd BD Z WARNING
AND NOT   D001340.B	// R_3rd BD Z MODULE ERR
AND NOT   D001340.C	// R_3rd BD Z SVD ERR
AND NOT   M00783	// R_3rd BD Z NOT MV
NOT
AND       M00008	// LEFT RESET SW PLS
ORP       T0918	// R_3rd BD Z LMT RST TM
OR        D002340.2	// R_3rd BD Z SERVO RESET
AND NOT   T0818	// R_3rd BD Z RST TM
OUT       D002340.2	// R_3rd BD Z SERVO RESET
TON       T0818 1	// R_3rd BD Z RST TM
; L122
LOAD      F00099
DMOV      D004882 D002348	// R_3rd BD Z A¢Ò¡¾¡¿Au¨ùO
// Currnent Postition
; L124
LOADD=    D004840 D001346
AND       T0518	// R_3rd_18 Z READY
AND       M01682	// R_3rd_18 Z HOME GOOD
OUT       M04180	// R_3rd_18 Z Pos.1st UP
; L125
LOADD=    D004842 D001346
AND       T0518	// R_3rd_18 Z READY
AND       M01682	// R_3rd_18 Z HOME GOOD
OUT       M04181	// R_3rd_18 Z Pos.2nd CENTER
; L126
LOADD=    D004844 D001346	// R_3rd BD Z BENDING POS
AND       T0518	// R_3rd_18 Z READY
AND       M01682	// R_3rd_18 Z HOME GOOD
AND NOT   M1902F	// DRY RUN
LOADD=    D004846 D001346
AND       T0518	// R_3rd_18 Z READY
AND       M01682	// R_3rd_18 Z HOME GOOD
AND       M1902F	// DRY RUN
OR LOAD
OUT       M04182	// R_3rd_18 Z Pos.3rd BEND.1st
; L128
LOAD      F00099
DADD      D004842 100 D004846
; L129
LOADD<    D004848 D004844	// R_3rd BD LIMIT / R_3rd BD Z BENDING POS
DMOV      D004848 D004844	// R_3rd BD LIMIT / R_3rd BD Z BENDING POS
// ----------------------------------------------------------------------------------
// 
// ----  < 19_R_2nd BENDING R >       SERVO MOTOR STATUS  HOME Search
// 
// ----------------------------------------------------------------------------------
; L131
LOAD      D001360.0	// R_2nd BD Z CTRL RDY
AND       D001360.2	// R_2nd BD Z SVD ON
AND NOT   D001360.6	// R_2nd BD Z SVD BUSY
AND NOT   D001360.A	// R_2nd BD Z WARNING
AND NOT   D001360.B	// R_2nd BD Z MODULE ERR
AND NOT   D001360.C	// R_2nd BD Z SVD ERR
AND NOT   M0169A	// L_2nd_19 R
AND NOT   M00783	// R_3rd BD Z NOT MV
AND NOT   M0169F	// L_2nd_19 R MOVE HOLD
OUT       M01690	// L_2nd_19 R READY

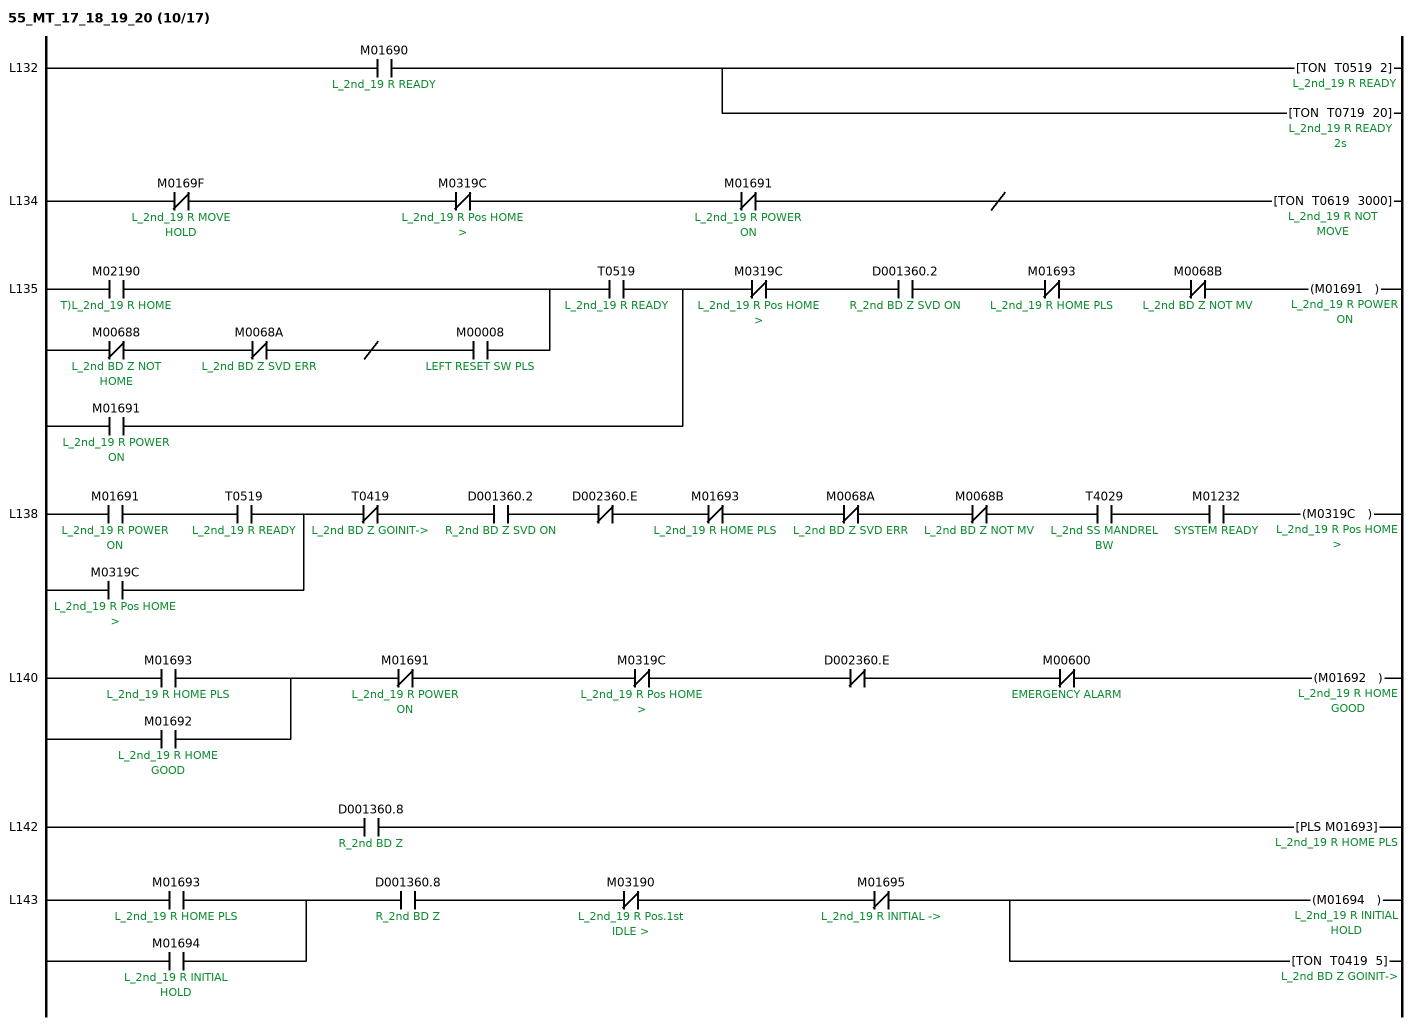
; L132
LOAD      M01690	// L_2nd_19 R READY
TON       T0519 2	// L_2nd_19 R READY
TON       T0719 20	// L_2nd_19 R READY 2s
; L134
LOAD NOT  M0169F	// L_2nd_19 R MOVE HOLD
AND NOT   M0319C	// L_2nd_19 R Pos HOME >
AND NOT   M01691	// L_2nd_19 R POWER ON
NOT
TON       T0619 3000	// L_2nd_19 R NOT MOVE
; L135
LOAD      M02190	// T)L_2nd_19 R HOME
LOAD NOT  M00688	// L_2nd BD Z NOT HOME
AND NOT   M0068A	// L_2nd BD Z SVD ERR
NOT
AND       M00008	// LEFT RESET SW PLS
OR LOAD
AND       T0519	// L_2nd_19 R READY
OR        M01691	// L_2nd_19 R POWER ON
AND NOT   M0319C	// L_2nd_19 R Pos HOME >
AND       D001360.2	// R_2nd BD Z SVD ON
AND NOT   M01693	// L_2nd_19 R HOME PLS
AND NOT   M0068B	// L_2nd BD Z NOT MV
OUT       M01691	// L_2nd_19 R POWER ON
; L138
LOAD      M01691	// L_2nd_19 R POWER ON
AND       T0519	// L_2nd_19 R READY
OR        M0319C	// L_2nd_19 R Pos HOME >
AND NOT   T0419	// L_2nd BD Z GOINIT->
AND       D001360.2	// R_2nd BD Z SVD ON
AND NOT   D002360.E
AND NOT   M01693	// L_2nd_19 R HOME PLS
AND NOT   M0068A	// L_2nd BD Z SVD ERR
AND NOT   M0068B	// L_2nd BD Z NOT MV
AND       T4029	// L_2nd SS MANDREL BW
AND       M01232	// SYSTEM READY
OUT       M0319C	// L_2nd_19 R Pos HOME >
; L140
LOAD      M01693	// L_2nd_19 R HOME PLS
OR        M01692	// L_2nd_19 R HOME GOOD
AND NOT   M01691	// L_2nd_19 R POWER ON
AND NOT   M0319C	// L_2nd_19 R Pos HOME >
AND NOT   D002360.E
AND NOT   M00600	// EMERGENCY ALARM
OUT       M01692	// L_2nd_19 R HOME GOOD
; L142
LOAD      D001360.8	// R_2nd BD Z
OUTP      M01693	// L_2nd_19 R HOME PLS
; L143
LOAD      M01693	// L_2nd_19 R HOME PLS
OR        M01694	// L_2nd_19 R INITIAL HOLD
AND       D001360.8	// R_2nd BD Z
AND NOT   M03190	// L_2nd_19 R Pos.1st IDLE >
AND NOT   M01695	// L_2nd_19 R INITIAL ->
OUT       M01694	// L_2nd_19 R INITIAL HOLD
TON       T0419 5	// L_2nd BD Z GOINIT->

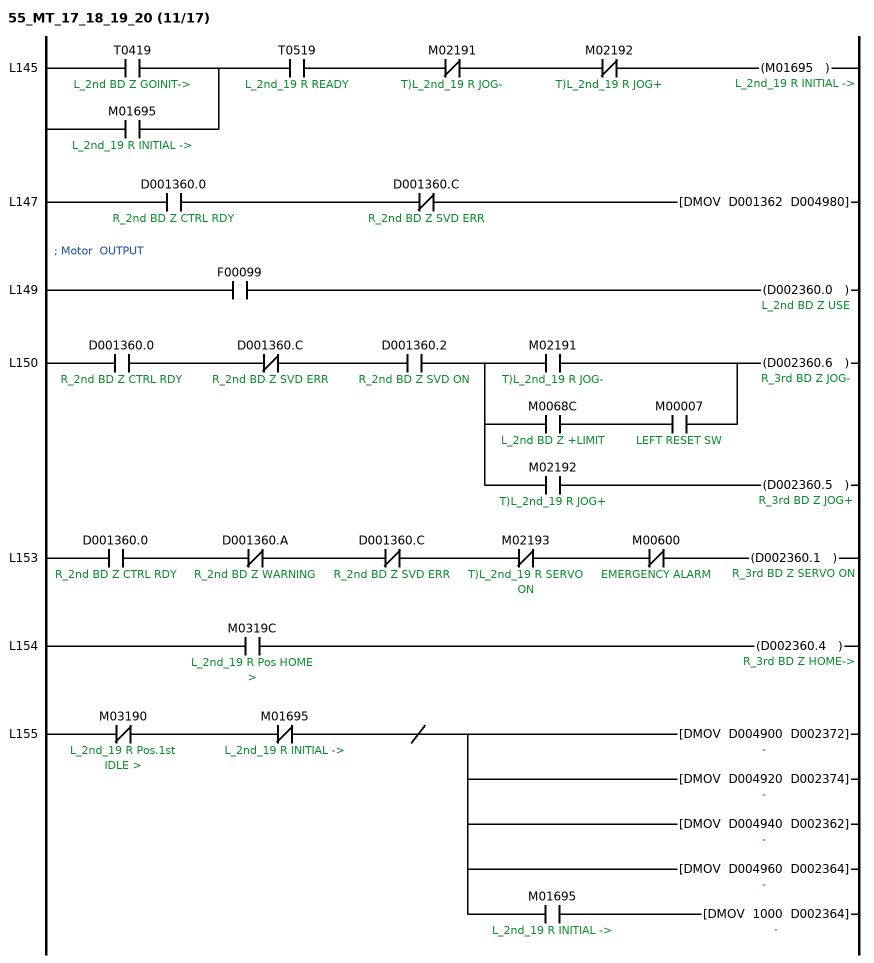
; L145
LOAD      T0419	// L_2nd BD Z GOINIT->
OR        M01695	// L_2nd_19 R INITIAL ->
AND       T0519	// L_2nd_19 R READY
AND NOT   M02191	// T)L_2nd_19 R JOG-
AND NOT   M02192	// T)L_2nd_19 R JOG+
OUT       M01695	// L_2nd_19 R INITIAL ->
; L147
LOAD      D001360.0	// R_2nd BD Z CTRL RDY
AND NOT   D001360.C	// R_2nd BD Z SVD ERR
DMOV      D001362 D004980
//  Motor  OUTPUT
; L149
LOAD      F00099
OUT       D002360.0	// L_2nd BD Z USE
; L150
LOAD      D001360.0	// R_2nd BD Z CTRL RDY
AND NOT   D001360.C	// R_2nd BD Z SVD ERR
AND       D001360.2	// R_2nd BD Z SVD ON
MPUSH
LOAD      M02191	// T)L_2nd_19 R JOG-
LOAD      M0068C	// L_2nd BD Z +LIMIT
AND       M00007	// LEFT RESET SW
OR LOAD
AND LOAD
OUT       D002360.6	// R_3rd BD Z JOG-
MPOP
AND       M02192	// T)L_2nd_19 R JOG+
OUT       D002360.5	// R_3rd BD Z JOG+
; L153
LOAD      D001360.0	// R_2nd BD Z CTRL RDY
AND NOT   D001360.A	// R_2nd BD Z WARNING
AND NOT   D001360.C	// R_2nd BD Z SVD ERR
AND NOT   M02193	// T)L_2nd_19 R SERVO ON
AND NOT   M00600	// EMERGENCY ALARM
OUT       D002360.1	// R_3rd BD Z SERVO ON
; L154
LOAD      M0319C	// L_2nd_19 R Pos HOME >
OUT       D002360.4	// R_3rd BD Z HOME->
; L155
LOAD NOT  M03190	// L_2nd_19 R Pos.1st IDLE >
AND NOT   M01695	// L_2nd_19 R INITIAL ->
NOT
DMOV      D004900 D002372	// -
DMOV      D004920 D002374	// -
DMOV      D004940 D002362	// -
DMOV      D004960 D002364	// -
AND       M01695	// L_2nd_19 R INITIAL ->
DMOV      1000 D002364	// -

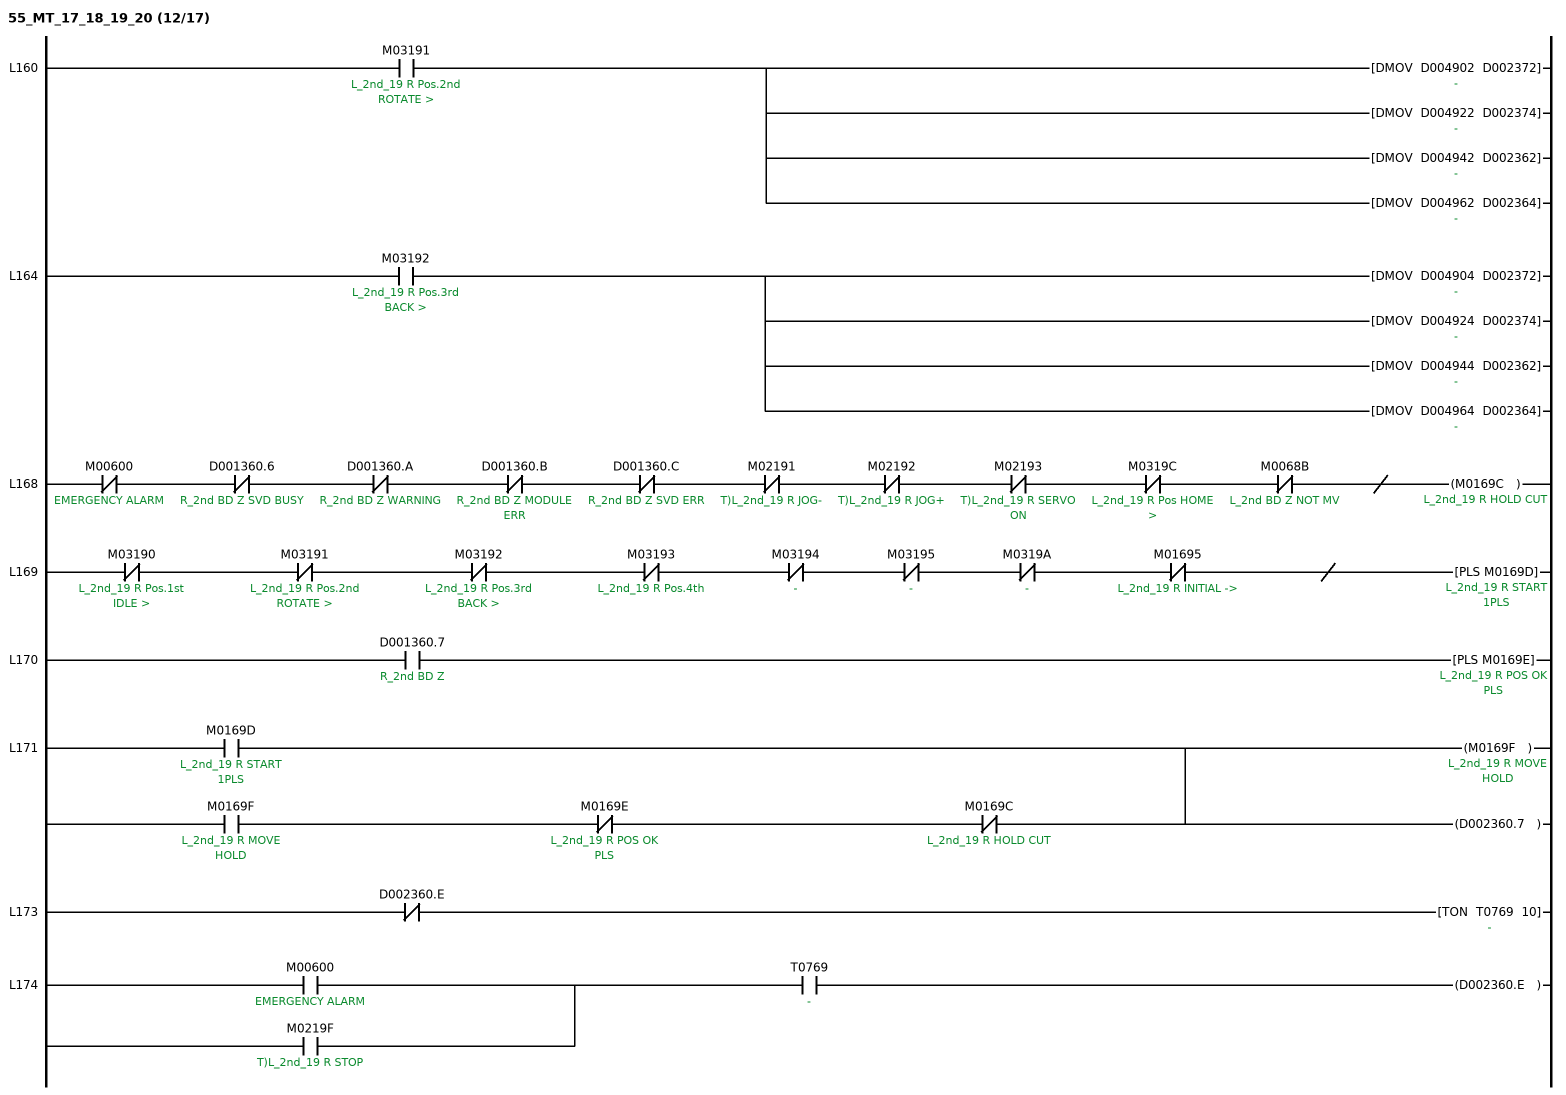
; L160
LOAD      M03191	// L_2nd_19 R Pos.2nd ROTATE >
DMOV      D004902 D002372	// -
DMOV      D004922 D002374	// -
DMOV      D004942 D002362	// -
DMOV      D004962 D002364	// -
; L164
LOAD      M03192	// L_2nd_19 R Pos.3rd BACK >
DMOV      D004904 D002372	// -
DMOV      D004924 D002374	// -
DMOV      D004944 D002362	// -
DMOV      D004964 D002364	// -
; L168
LOAD NOT  M00600	// EMERGENCY ALARM
AND NOT   D001360.6	// R_2nd BD Z SVD BUSY
AND NOT   D001360.A	// R_2nd BD Z WARNING
AND NOT   D001360.B	// R_2nd BD Z MODULE ERR
AND NOT   D001360.C	// R_2nd BD Z SVD ERR
AND NOT   M02191	// T)L_2nd_19 R JOG-
AND NOT   M02192	// T)L_2nd_19 R JOG+
AND NOT   M02193	// T)L_2nd_19 R SERVO ON
AND NOT   M0319C	// L_2nd_19 R Pos HOME >
AND NOT   M0068B	// L_2nd BD Z NOT MV
NOT
OUT       M0169C	// L_2nd_19 R HOLD CUT
; L169
LOAD NOT  M03190	// L_2nd_19 R Pos.1st IDLE >
AND NOT   M03191	// L_2nd_19 R Pos.2nd ROTATE >
AND NOT   M03192	// L_2nd_19 R Pos.3rd BACK >
AND NOT   M03193	// L_2nd_19 R Pos.4th 
AND NOT   M03194	// -
AND NOT   M03195	// -
AND NOT   M0319A	// -
AND NOT   M01695	// L_2nd_19 R INITIAL ->
NOT
OUTP      M0169D	// L_2nd_19 R START 1PLS
; L170
LOAD      D001360.7	// R_2nd BD Z
OUTP      M0169E	// L_2nd_19 R POS OK PLS
; L171
LOAD      M0169D	// L_2nd_19 R START 1PLS
LOAD      M0169F	// L_2nd_19 R MOVE HOLD
AND NOT   M0169E	// L_2nd_19 R POS OK PLS
AND NOT   M0169C	// L_2nd_19 R HOLD CUT
OR LOAD
OUT       M0169F	// L_2nd_19 R MOVE HOLD
OUT       D002360.7
; L173
LOAD NOT  D002360.E
TON       T0769 10	// -
; L174
LOAD      M00600	// EMERGENCY ALARM
OR        M0219F	// T)L_2nd_19 R STOP
AND       T0769	// -
OUT       D002360.E

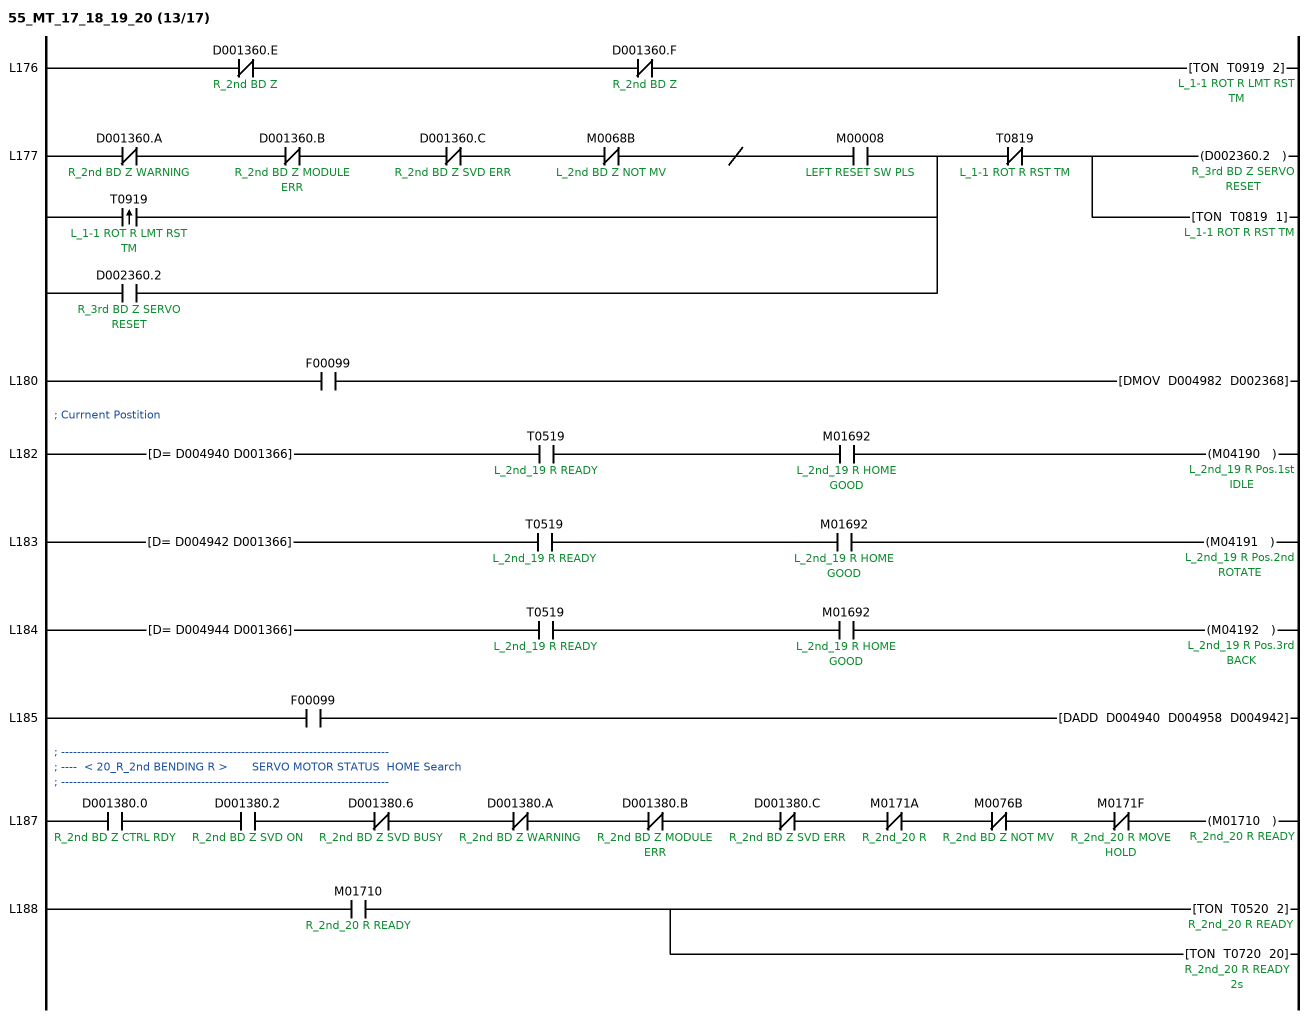
; L176
LOAD NOT  D001360.E	// R_2nd BD Z
AND NOT   D001360.F	// R_2nd BD Z
TON       T0919 2	// L_1-1 ROT R LMT RST TM
; L177
LOAD NOT  D001360.A	// R_2nd BD Z WARNING
AND NOT   D001360.B	// R_2nd BD Z MODULE ERR
AND NOT   D001360.C	// R_2nd BD Z SVD ERR
AND NOT   M0068B	// L_2nd BD Z NOT MV
NOT
AND       M00008	// LEFT RESET SW PLS
ORP       T0919	// L_1-1 ROT R LMT RST TM
OR        D002360.2	// R_3rd BD Z SERVO RESET
AND NOT   T0819	// L_1-1 ROT R RST TM
OUT       D002360.2	// R_3rd BD Z SERVO RESET
TON       T0819 1	// L_1-1 ROT R RST TM
; L180
LOAD      F00099
DMOV      D004982 D002368
// Currnent Postition
; L182
LOADD=    D004940 D001366
AND       T0519	// L_2nd_19 R READY
AND       M01692	// L_2nd_19 R HOME GOOD
OUT       M04190	// L_2nd_19 R Pos.1st IDLE
; L183
LOADD=    D004942 D001366
AND       T0519	// L_2nd_19 R READY
AND       M01692	// L_2nd_19 R HOME GOOD
OUT       M04191	// L_2nd_19 R Pos.2nd ROTATE
; L184
LOADD=    D004944 D001366
AND       T0519	// L_2nd_19 R READY
AND       M01692	// L_2nd_19 R HOME GOOD
OUT       M04192	// L_2nd_19 R Pos.3rd BACK
; L185
LOAD      F00099
DADD      D004940 D004958 D004942
// ----------------------------------------------------------------------------------
// 
// ----  < 20_R_2nd BENDING R >       SERVO MOTOR STATUS  HOME Search
// 
// ----------------------------------------------------------------------------------
; L187
LOAD      D001380.0	// R_2nd BD Z CTRL RDY
AND       D001380.2	// R_2nd BD Z SVD ON
AND NOT   D001380.6	// R_2nd BD Z SVD BUSY
AND NOT   D001380.A	// R_2nd BD Z WARNING
AND NOT   D001380.B	// R_2nd BD Z MODULE ERR
AND NOT   D001380.C	// R_2nd BD Z SVD ERR
AND NOT   M0171A	// R_2nd_20 R
AND NOT   M0076B	// R_2nd BD Z NOT MV
AND NOT   M0171F	// R_2nd_20 R MOVE HOLD
OUT       M01710	// R_2nd_20 R READY
; L188
LOAD      M01710	// R_2nd_20 R READY
TON       T0520 2	// R_2nd_20 R READY
TON       T0720 20	// R_2nd_20 R READY 2s

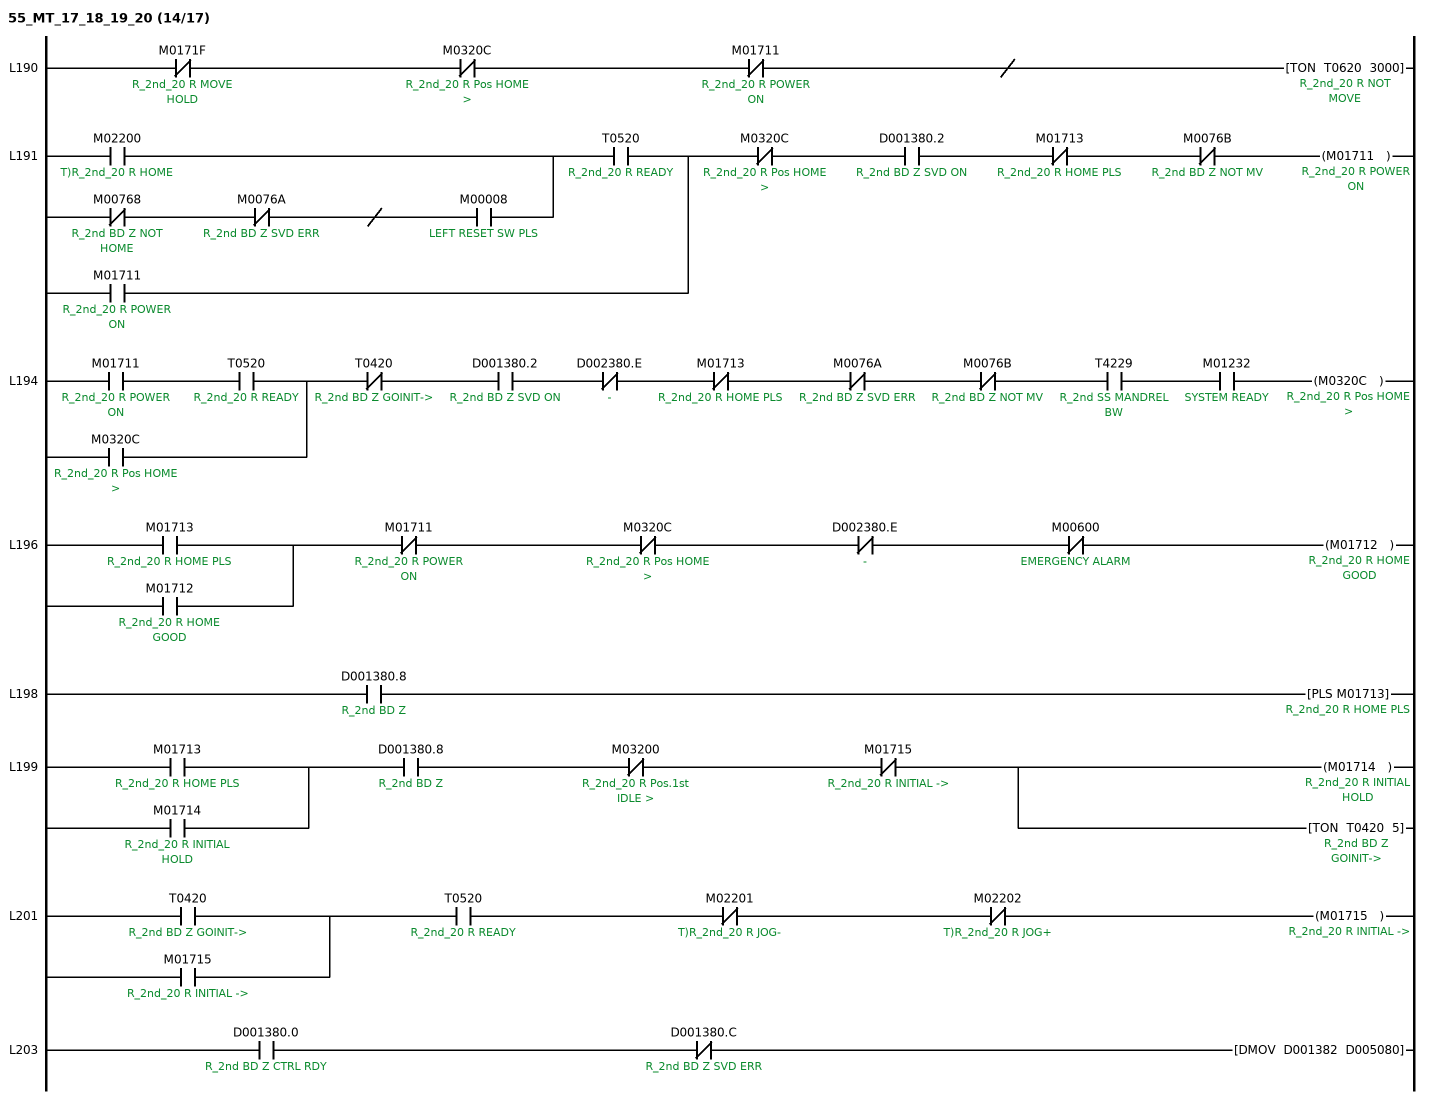
; L190
LOAD NOT  M0171F	// R_2nd_20 R MOVE HOLD
AND NOT   M0320C	// R_2nd_20 R Pos HOME >
AND NOT   M01711	// R_2nd_20 R POWER ON
NOT
TON       T0620 3000	// R_2nd_20 R NOT MOVE
; L191
LOAD      M02200	// T)R_2nd_20 R HOME
LOAD NOT  M00768	// R_2nd BD Z NOT HOME
AND NOT   M0076A	// R_2nd BD Z SVD ERR
NOT
AND       M00008	// LEFT RESET SW PLS
OR LOAD
AND       T0520	// R_2nd_20 R READY
OR        M01711	// R_2nd_20 R POWER ON
AND NOT   M0320C	// R_2nd_20 R Pos HOME >
AND       D001380.2	// R_2nd BD Z SVD ON
AND NOT   M01713	// R_2nd_20 R HOME PLS
AND NOT   M0076B	// R_2nd BD Z NOT MV
OUT       M01711	// R_2nd_20 R POWER ON
; L194
LOAD      M01711	// R_2nd_20 R POWER ON
AND       T0520	// R_2nd_20 R READY
OR        M0320C	// R_2nd_20 R Pos HOME >
AND NOT   T0420	// R_2nd BD Z GOINIT->
AND       D001380.2	// R_2nd BD Z SVD ON
AND NOT   D002380.E	// -
AND NOT   M01713	// R_2nd_20 R HOME PLS
AND NOT   M0076A	// R_2nd BD Z SVD ERR
AND NOT   M0076B	// R_2nd BD Z NOT MV
AND       T4229	// R_2nd SS MANDREL BW
AND       M01232	// SYSTEM READY
OUT       M0320C	// R_2nd_20 R Pos HOME >
; L196
LOAD      M01713	// R_2nd_20 R HOME PLS
OR        M01712	// R_2nd_20 R HOME GOOD
AND NOT   M01711	// R_2nd_20 R POWER ON
AND NOT   M0320C	// R_2nd_20 R Pos HOME >
AND NOT   D002380.E	// -
AND NOT   M00600	// EMERGENCY ALARM
OUT       M01712	// R_2nd_20 R HOME GOOD
; L198
LOAD      D001380.8	// R_2nd BD Z
OUTP      M01713	// R_2nd_20 R HOME PLS
; L199
LOAD      M01713	// R_2nd_20 R HOME PLS
OR        M01714	// R_2nd_20 R INITIAL HOLD
AND       D001380.8	// R_2nd BD Z
AND NOT   M03200	// R_2nd_20 R Pos.1st IDLE >
AND NOT   M01715	// R_2nd_20 R INITIAL ->
OUT       M01714	// R_2nd_20 R INITIAL HOLD
TON       T0420 5	// R_2nd BD Z GOINIT->
; L201
LOAD      T0420	// R_2nd BD Z GOINIT->
OR        M01715	// R_2nd_20 R INITIAL ->
AND       T0520	// R_2nd_20 R READY
AND NOT   M02201	// T)R_2nd_20 R JOG-
AND NOT   M02202	// T)R_2nd_20 R JOG+
OUT       M01715	// R_2nd_20 R INITIAL ->
; L203
LOAD      D001380.0	// R_2nd BD Z CTRL RDY
AND NOT   D001380.C	// R_2nd BD Z SVD ERR
DMOV      D001382 D005080

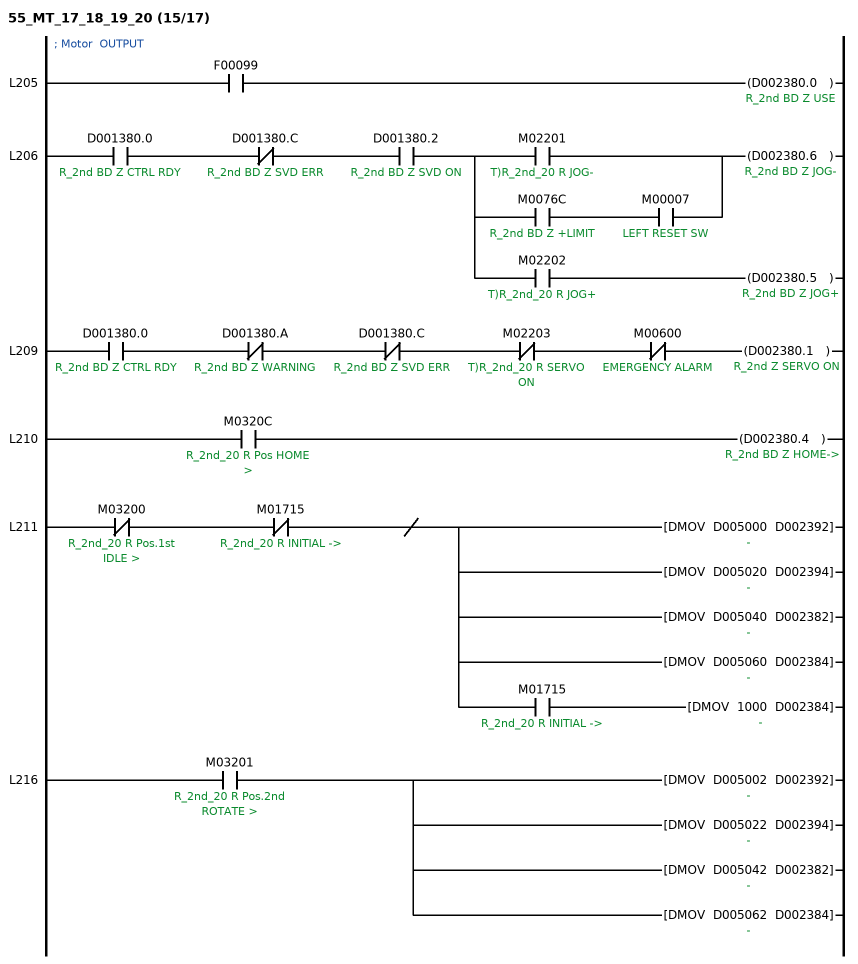
//  Motor  OUTPUT
; L205
LOAD      F00099
OUT       D002380.0	// R_2nd BD Z USE
; L206
LOAD      D001380.0	// R_2nd BD Z CTRL RDY
AND NOT   D001380.C	// R_2nd BD Z SVD ERR
AND       D001380.2	// R_2nd BD Z SVD ON
MPUSH
LOAD      M02201	// T)R_2nd_20 R JOG-
LOAD      M0076C	// R_2nd BD Z +LIMIT
AND       M00007	// LEFT RESET SW
OR LOAD
AND LOAD
OUT       D002380.6	// R_2nd BD Z JOG-
MPOP
AND       M02202	// T)R_2nd_20 R JOG+
OUT       D002380.5	// R_2nd BD Z JOG+
; L209
LOAD      D001380.0	// R_2nd BD Z CTRL RDY
AND NOT   D001380.A	// R_2nd BD Z WARNING
AND NOT   D001380.C	// R_2nd BD Z SVD ERR
AND NOT   M02203	// T)R_2nd_20 R SERVO ON
AND NOT   M00600	// EMERGENCY ALARM
OUT       D002380.1	// R_2nd Z SERVO ON
; L210
LOAD      M0320C	// R_2nd_20 R Pos HOME >
OUT       D002380.4	// R_2nd BD Z HOME->
; L211
LOAD NOT  M03200	// R_2nd_20 R Pos.1st IDLE >
AND NOT   M01715	// R_2nd_20 R INITIAL ->
NOT
DMOV      D005000 D002392	// -
DMOV      D005020 D002394	// -
DMOV      D005040 D002382	// -
DMOV      D005060 D002384	// -
AND       M01715	// R_2nd_20 R INITIAL ->
DMOV      1000 D002384	// -
; L216
LOAD      M03201	// R_2nd_20 R Pos.2nd ROTATE >
DMOV      D005002 D002392	// -
DMOV      D005022 D002394	// -
DMOV      D005042 D002382	// -
DMOV      D005062 D002384	// -

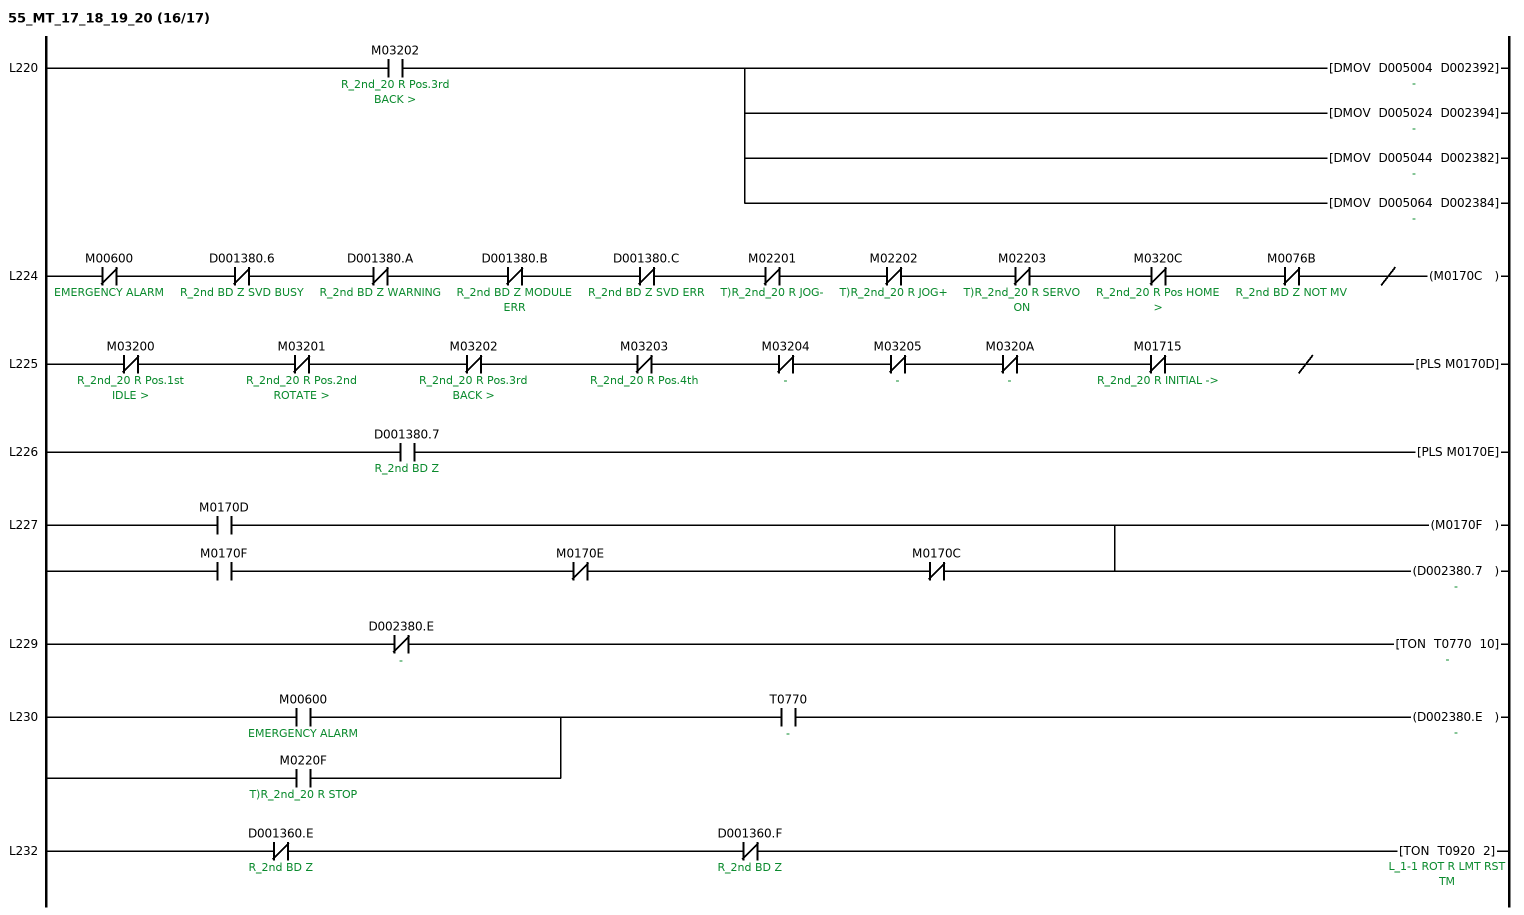
; L220
LOAD      M03202	// R_2nd_20 R Pos.3rd BACK >
DMOV      D005004 D002392	// -
DMOV      D005024 D002394	// -
DMOV      D005044 D002382	// -
DMOV      D005064 D002384	// -
; L224
LOAD NOT  M00600	// EMERGENCY ALARM
AND NOT   D001380.6	// R_2nd BD Z SVD BUSY
AND NOT   D001380.A	// R_2nd BD Z WARNING
AND NOT   D001380.B	// R_2nd BD Z MODULE ERR
AND NOT   D001380.C	// R_2nd BD Z SVD ERR
AND NOT   M02201	// T)R_2nd_20 R JOG-
AND NOT   M02202	// T)R_2nd_20 R JOG+
AND NOT   M02203	// T)R_2nd_20 R SERVO ON
AND NOT   M0320C	// R_2nd_20 R Pos HOME >
AND NOT   M0076B	// R_2nd BD Z NOT MV
NOT
OUT       M0170C
; L225
LOAD NOT  M03200	// R_2nd_20 R Pos.1st IDLE >
AND NOT   M03201	// R_2nd_20 R Pos.2nd ROTATE >
AND NOT   M03202	// R_2nd_20 R Pos.3rd BACK >
AND NOT   M03203	// R_2nd_20 R Pos.4th 
AND NOT   M03204	// -
AND NOT   M03205	// -
AND NOT   M0320A	// -
AND NOT   M01715	// R_2nd_20 R INITIAL ->
NOT
OUTP      M0170D
; L226
LOAD      D001380.7	// R_2nd BD Z
OUTP      M0170E
; L227
LOAD      M0170D
LOAD      M0170F
AND NOT   M0170E
AND NOT   M0170C
OR LOAD
OUT       M0170F
OUT       D002380.7	// -
; L229
LOAD NOT  D002380.E	// -
TON       T0770 10	// -
; L230
LOAD      M00600	// EMERGENCY ALARM
OR        M0220F	// T)R_2nd_20 R STOP
AND       T0770	// -
OUT       D002380.E	// -
; L232
LOAD NOT  D001360.E	// R_2nd BD Z
AND NOT   D001360.F	// R_2nd BD Z
TON       T0920 2	// L_1-1 ROT R LMT RST TM

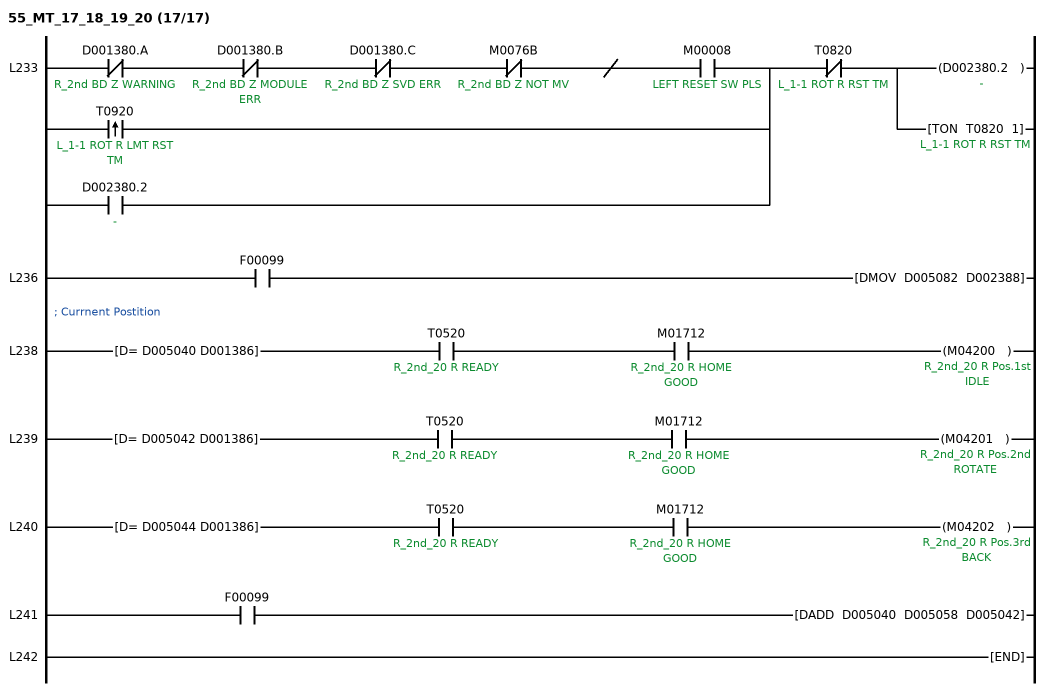
; L233
LOAD NOT  D001380.A	// R_2nd BD Z WARNING
AND NOT   D001380.B	// R_2nd BD Z MODULE ERR
AND NOT   D001380.C	// R_2nd BD Z SVD ERR
AND NOT   M0076B	// R_2nd BD Z NOT MV
NOT
AND       M00008	// LEFT RESET SW PLS
ORP       T0920	// L_1-1 ROT R LMT RST TM
OR        D002380.2	// -
AND NOT   T0820	// L_1-1 ROT R RST TM
OUT       D002380.2	// -
TON       T0820 1	// L_1-1 ROT R RST TM
; L236
LOAD      F00099
DMOV      D005082 D002388
// Currnent Postition
; L238
LOADD=    D005040 D001386
AND       T0520	// R_2nd_20 R READY
AND       M01712	// R_2nd_20 R HOME GOOD
OUT       M04200	// R_2nd_20 R Pos.1st IDLE
; L239
LOADD=    D005042 D001386
AND       T0520	// R_2nd_20 R READY
AND       M01712	// R_2nd_20 R HOME GOOD
OUT       M04201	// R_2nd_20 R Pos.2nd ROTATE
; L240
LOADD=    D005044 D001386
AND       T0520	// R_2nd_20 R READY
AND       M01712	// R_2nd_20 R HOME GOOD
OUT       M04202	// R_2nd_20 R Pos.3rd BACK
; L241
LOAD      F00099
DADD      D005040 D005058 D005042
; L242
END

PROGRAM 81_OUTPUT (task: ¨ö¨¬A¥ì CA¡¤I¡¾¡¿¡¤¡Í)

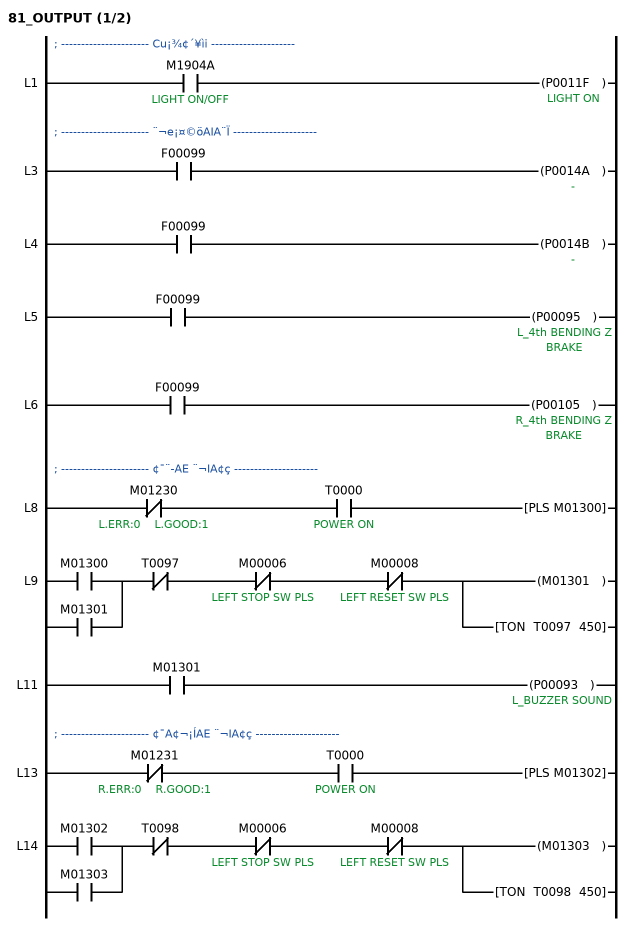
// ---------------------- Cu¡¾¢´¥ìi ---------------------
; L1
LOAD      M1904A	// LIGHT ON/OFF
OUT       P0011F	// LIGHT ON
// ---------------------- ¨¬e¡¤©öAIA¨Ï ---------------------
; L3
LOAD      F00099
OUT       P0014A	// -
; L4
LOAD      F00099
OUT       P0014B	// -
; L5
LOAD      F00099
OUT       P00095	// L_4th BENDING Z BRAKE
; L6
LOAD      F00099
OUT       P00105	// R_4th BENDING Z BRAKE
// ---------------------- ¢¯¨­AE ¨¬IA¢ç ---------------------
; L8
LOAD NOT  M01230	// L.ERR:0    L.GOOD:1
AND       T0000	// POWER ON
OUTP      M01300
; L9
LOAD      M01300
OR        M01301
AND NOT   T0097
AND NOT   M00006	// LEFT STOP SW PLS
AND NOT   M00008	// LEFT RESET SW PLS
OUT       M01301
TON       T0097 450
; L11
LOAD      M01301
OUT       P00093	// L_BUZZER SOUND
// ---------------------- ¢¯A¢¬¡ÍAE ¨¬IA¢ç ---------------------
; L13
LOAD NOT  M01231	// R.ERR:0    R.GOOD:1
AND       T0000	// POWER ON
OUTP      M01302
; L14
LOAD      M01302
OR        M01303
AND NOT   T0098
AND NOT   M00006	// LEFT STOP SW PLS
AND NOT   M00008	// LEFT RESET SW PLS
OUT       M01303
TON       T0098 450

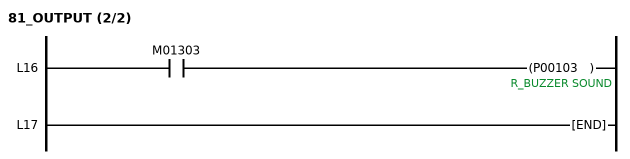
; L16
LOAD      M01303
OUT       P00103	// R_BUZZER SOUND
; L17
END

PROGRAM 82_L_MANUAL (task: ¨ö¨¬A¥ì CA¡¤I¡¾¡¿¡¤¡Í)

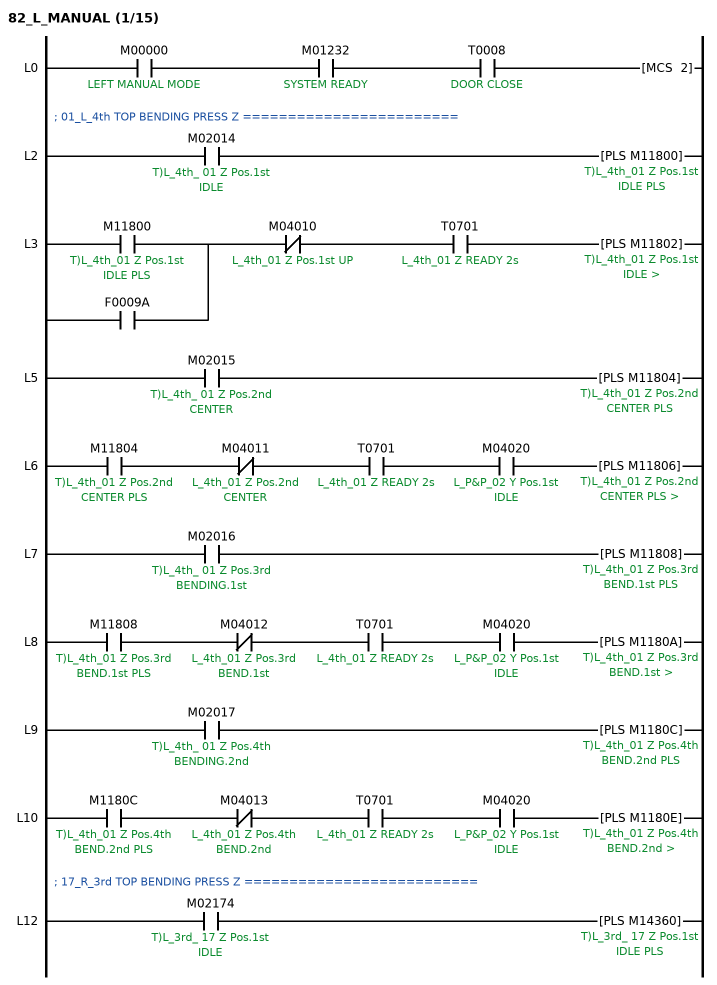
; L0
LOAD      M00000	// LEFT MANUAL MODE
AND       M01232	// SYSTEM READY
AND       T0008	// DOOR CLOSE
MCS       2
// 01_L_4th TOP BENDING PRESS Z ======================== 
; L2
LOAD      M02014	// T)L_4th_ 01 Z Pos.1st IDLE
OUTP      M11800	// T)L_4th_01 Z Pos.1st IDLE PLS
; L3
LOAD      M11800	// T)L_4th_01 Z Pos.1st IDLE PLS
OR        F0009A
AND NOT   M04010	// L_4th_01 Z Pos.1st UP
AND       T0701	// L_4th_01 Z READY 2s
OUTP      M11802	// T)L_4th_01 Z Pos.1st IDLE >
; L5
LOAD      M02015	// T)L_4th_ 01 Z Pos.2nd CENTER
OUTP      M11804	// T)L_4th_01 Z Pos.2nd CENTER PLS
; L6
LOAD      M11804	// T)L_4th_01 Z Pos.2nd CENTER PLS
AND NOT   M04011	// L_4th_01 Z Pos.2nd CENTER
AND       T0701	// L_4th_01 Z READY 2s
AND       M04020	// L_P&P_02 Y Pos.1st IDLE
OUTP      M11806	// T)L_4th_01 Z Pos.2nd CENTER PLS >
; L7
LOAD      M02016	// T)L_4th_ 01 Z Pos.3rd BENDING.1st
OUTP      M11808	// T)L_4th_01 Z Pos.3rd BEND.1st PLS
; L8
LOAD      M11808	// T)L_4th_01 Z Pos.3rd BEND.1st PLS
AND NOT   M04012	// L_4th_01 Z Pos.3rd BEND.1st
AND       T0701	// L_4th_01 Z READY 2s
AND       M04020	// L_P&P_02 Y Pos.1st IDLE
OUTP      M1180A	// T)L_4th_01 Z Pos.3rd BEND.1st >
; L9
LOAD      M02017	// T)L_4th_ 01 Z Pos.4th BENDING.2nd
OUTP      M1180C	// T)L_4th_01 Z Pos.4th BEND.2nd PLS
; L10
LOAD      M1180C	// T)L_4th_01 Z Pos.4th BEND.2nd PLS
AND NOT   M04013	// L_4th_01 Z Pos.4th BEND.2nd
AND       T0701	// L_4th_01 Z READY 2s
AND       M04020	// L_P&P_02 Y Pos.1st IDLE
OUTP      M1180E	// T)L_4th_01 Z Pos.4th BEND.2nd >
// 17_R_3rd TOP BENDING PRESS Z ==========================
; L12
LOAD      M02174	// T)L_3rd_ 17 Z Pos.1st IDLE
OUTP      M14360	// T)L_3rd_ 17 Z Pos.1st IDLE PLS

